Yaskawa INFORM job: SKRZYNIA_5540_90_STOPNI_10BR.JBI

/JOB
//NAME SKRZYNIA_5540_90_STOPNI_10BR
///FOLDERNAME 02-SKRZYNIE_JOBS
//POS
///NPOS 687,687,0,50,0,0
///TOOL 0
///POSTYPE PULSE
///PULSE
C00000=0,-52280,40443,0,6876,0
C00001=82314,-24956,17040,59626,-27382,6248
C00002=93910,-8625,17040,59626,-43355,6248
C00003=98846,-1061,-42166,80308,-57081,-16120
C00004=100452,6057,-48127,85711,-56704,-21322
C00005=96349,29000,-36127,85072,-63022,-26262
C00006=95580,33075,-33256,84644,-64024,-26851
C00007=94197,33846,-32020,85210,-63413,-26698
C00008=95580,33075,-33256,84644,-64024,-26851
C00009=94888,31114,-36362,85298,-63687,-27185
C00010=95580,33075,-33256,84644,-64024,-26851
C00011=95263,33142,-33256,84677,-63995,-26850
C00012=94634,33491,-32695,84935,-63717,-26781
C00013=94130,33776,-32235,85140,-63494,-26725
C00014=95104,32689,-33981,84829,-63917,-26928
C00015=94679,31503,-35865,85229,-63711,-27129
C00016=95263,33142,-33256,84677,-63995,-26850
C00017=95260,33144,-33256,84678,-63995,-26850
C00018=94650,33483,-32714,84929,-63727,-26783
C00019=94112,33789,-32223,85148,-63489,-26723
C00020=95084,32644,-34054,84845,-63909,-26937
C00021=94657,31449,-35950,85247,-63703,-27139
C00022=95260,33144,-33256,84678,-63995,-26850
C00023=95258,33145,-33257,84676,-63996,-26846
C00024=94953,33314,-32988,84801,-63862,-26812
C00025=94037,33833,-32158,85174,-63457,-26709
C00026=94978,32352,-34521,84941,-63860,-26983
C00027=94597,31295,-36193,85297,-63678,-27162
C00028=95258,33145,-33257,84676,-63996,-26846
C00029=95258,33145,-33257,84676,-63996,-26846
C00030=94635,33491,-32703,84932,-63720,-26777
C00031=94255,33706,-32357,85087,-63552,-26734
C00032=95076,32627,-34084,84849,-63906,-26937
C00033=94616,31344,-36119,85281,-63684,-27155
C00034=95258,33145,-33257,84676,-63996,-26846
C00035=95258,25631,32269,66559,-75499,-2416
C00036=95045,25799,32513,66531,-75379,-2372
C00037=94321,26382,33365,66429,-74973,-2219
C00038=95048,24784,31042,66584,-75290,-2483
C00039=94601,23046,28557,66633,-74859,-2609
C00040=95258,25631,32269,66559,-75499,-2416
C00041=98646,19496,-17631,99827,-80462,-21224
C00042=98317,21326,-15127,99395,-81089,-20992
C00043=97962,21529,-14845,99504,-80870,-20995
C00044=98567,20146,-16748,99341,-81286,-21080
C00045=98203,18829,-18537,99489,-81121,-21211
C00046=98811,21047,-15512,99242,-81394,-20987
C00047=98811,19937,1242,97498,-78933,-15296
C00048=98811,19937,1242,97498,-78933,-15296
C00049=98014,20416,1894,97635,-78400,-15298
C00050=98593,19084,88,97564,-78819,-15379
C00051=98194,17557,-1953,97683,-78607,-15521
C00052=98811,19937,1242,97498,-78933,-15296
C00053=98765,34858,63506,90961,-74847,-417
C00054=98962,39103,70654,91062,-76265,452
C00055=98093,40155,72476,90768,-75677,655
C00056=98962,39103,70654,91062,-76265,452
C00057=98539,36034,65455,91246,-76081,-158
C00058=98962,39103,70654,91062,-76265,452
C00059=98994,31803,58419,90917,-73461,-1055
C00060=94428,854,16076,89248,-50738,-4740
C00061=88080,-20128,-3199,80943,-31244,-2335
C00062=48287,-44591,-17414,16172,-14532,25809
C00063=48287,-44591,-17414,16172,-14532,25809
C00064=89603,-12372,12158,50295,-44413,5810
C00065=98990,20110,21695,70166,-74669,-10293
C00066=97443,24182,16559,71706,-75040,-13643
C00067=96724,24681,12603,72193,-76238,-15336
C00068=95373,25645,13977,72253,-75425,-15117
C00069=96724,24681,12603,72193,-76238,-15336
C00070=96395,23390,10778,72281,-75950,-15438
C00071=96724,24681,12603,72193,-76238,-15336
C00072=98418,23275,9051,78885,-77594,-17480
C00073=98418,23353,9846,78794,-77668,-17252
C00074=97172,24175,11002,78894,-76868,-17107
C00075=98418,23353,9846,78794,-77668,-17252
C00076=98085,21992,7947,78885,-77405,-17367
C00077=98418,23353,9846,78794,-77668,-17252
C00078=97055,28839,36684,71776,-79389,-10554
C00079=97055,28839,36684,71776,-79389,-10554
C00080=96073,29634,37879,71669,-78808,-10363
C00081=97055,28839,36684,71776,-79389,-10554
C00082=96556,26588,33346,71835,-78895,-10784
C00083=97055,28839,36684,71776,-79389,-10554
C00084=97055,28839,36684,71776,-79389,-10554
C00085=97055,28839,36684,71776,-79389,-10554
C00086=96070,29634,37881,71667,-78806,-10365
C00087=97055,28839,36684,71776,-79389,-10554
C00088=96542,26531,33264,71837,-78884,-10788
C00089=97055,28839,36684,71776,-79389,-10554
C00090=99222,23346,17795,82202,-78388,4176
C00091=99222,23346,17795,82202,-78388,4176
C00092=98198,24012,18735,82231,-77709,4276
C00093=99222,23346,17795,82202,-78388,4176
C00094=98846,21740,15549,82282,-78105,4028
C00095=99222,23346,17795,82202,-78388,4176
C00096=97305,19304,15511,100837,-75687,4760
C00097=97826,25373,24000,100195,-79238,5786
C00098=96887,26043,24967,100223,-78578,5793
C00099=97826,25373,24000,100195,-79238,5786
C00100=97448,23764,21701,100276,-79072,5588
C00101=97826,25373,24000,100195,-79238,5786
C00102=97826,25373,24000,100195,-79238,5786
C00103=97826,25373,24000,100195,-79238,5786
C00104=96843,26076,25015,100223,-78545,5791
C00105=97826,25373,24000,100195,-79238,5786
C00106=97441,23730,21652,100278,-79068,5583
C00107=97826,25373,24000,100195,-79238,5786
C00108=98604,24841,23235,100170,-79782,5786
C00109=98281,23602,18484,100238,-79492,4693
C00110=96938,24614,19922,100310,-78605,4704
C00111=98281,23602,18484,100238,-79492,4693
C00112=97922,22110,16391,100318,-79328,4520
C00113=98281,23602,18484,100238,-79492,4693
C00114=97826,25373,24000,100195,-79238,5786
C00115=100071,8792,-2363,102947,-71408,2025
C00116=90699,-12620,-30080,113827,-52438,-6201
C00117=97832,-16290,-36993,112551,-57584,-6005
C00118=83036,-26396,-56580,138157,-49269,-16960
C00119=83036,-26453,-52828,136768,-47205,-15962
C00120=60067,-65836,-77869,147206,-28305,-20439
C00121=63330,-26972,24478,18707,-56801,31483
C00122=86830,-18603,-3985,49492,-42347,15253
C00123=100465,-3562,-10252,69901,-61773,-201
C00124=99635,18997,3540,80919,-74698,-6325
C00125=98097,22561,8426,80415,-76730,-6116
C00126=98097,22561,8426,80415,-76730,-6116
C00127=97377,23028,9077,80478,-76265,-6042
C00128=98097,22561,8426,80415,-76730,-6116
C00129=97807,21406,6827,80497,-76510,-6215
C00130=98097,22561,8426,80415,-76730,-6116
C00131=98919,31293,46565,87609,-78984,1304
C00132=98899,30801,44624,87834,-79065,838
C00133=98247,31325,45433,87747,-78622,912
C00134=98899,30801,44624,87834,-79065,838
C00135=98602,29264,42279,87883,-78869,621
C00136=98899,30801,44624,87834,-79065,838
C00137=98482,30562,41503,101958,-78355,-2440
C00138=98031,30614,41582,101940,-78055,-2471
C00139=96674,31741,43313,101828,-77074,-2426
C00140=98031,30614,41582,101940,-78055,-2471
C00141=97723,29096,39278,102008,-77969,-2698
C00142=98031,30614,41582,101940,-78055,-2471
C00143=99865,12124,7354,104364,-73625,-7862
C00144=80898,-21381,-5865,68721,-28456,7693
C00145=53207,-50775,-37673,21053,-11333,28727
C00146=44299,-51091,-32799,-7549,-14278,41753
///LIMIT ON
C00147=42754,-66126,12236,-1301,3231,7194
///LIMIT OFF
C00148=0,-52280,40443,0,6876,0
C00149=0,-52280,40443,0,6876,0
C00150=0,-43112,23163,-32261,-40956,-29092
C00151=48283,-21883,28214,25170,-26491,-48363
C00152=46664,-3144,58041,18842,-32105,-45325
C00153=50347,-18571,12268,49104,-16423,-60029
C00154=51149,-18702,10839,52647,-16284,-61663
C00155=49023,-16654,12458,50505,-14948,-60880
C00156=50458,-16314,12735,52976,-15639,-61913
C00157=50509,-19000,10610,51503,-15997,-61182
C00158=50509,-19000,10610,51503,-15997,-61182
C00159=51153,-18191,11234,52953,-16222,-61812
C00160=49506,-16603,12499,51322,-15186,-61219
C00161=50699,-16390,12671,53298,-15774,-62041
C00162=50704,-18403,11069,52157,-16018,-61478
C00163=50704,-18403,11069,52157,-16018,-61478
C00164=51011,-18259,11181,52703,-16157,-61707
C00165=49372,-16676,12437,51065,-15128,-61110
C00166=50855,-16321,12727,53567,-15849,-62152
C00167=50704,-18403,11069,52157,-16018,-61478
C00168=50704,-18403,11069,52157,-16018,-61478
C00169=51194,-17966,11787,52443,-16367,-61556
C00170=49641,-16469,12982,50879,-15396,-60984
C00171=51159,-16110,13274,53409,-16135,-62034
C00172=51194,-19029,8982,55593,-15729,-63095
C00173=51005,-17995,11387,52847,-16122,-61778
C00174=51030,-17982,11395,52891,-16135,-61798
C00175=49666,-16664,12446,51542,-15278,-61306
C00176=51234,-16283,12753,54139,-16047,-62382
C00177=51030,-17982,11395,52891,-16135,-61798
C00178=51030,-17982,11395,52891,-16135,-61798
C00179=51056,-17951,11420,52949,-16145,-61823
C00180=49507,-16445,12622,51407,-15172,-61259
C00181=51212,-15994,12989,54262,-16005,-62444
C00182=51056,-17951,11420,52949,-16145,-61823
C00183=50945,-18019,11363,52741,-16103,-61737
C00184=51451,-18380,9957,55416,-15976,-62984
C00185=49638,-16617,11364,53777,-14815,-62399
C00186=51249,-16205,11700,56405,-15635,-63491
C00187=50945,-18019,11363,52741,-16103,-61737
C00188=50945,-18019,11363,52741,-16103,-61737
C00189=51751,-18888,8325,57986,-15754,-64205
C00190=49901,-17096,9744,56519,-14545,-63700
C00191=51443,-16713,10055,58931,-15359,-64698
C00192=50945,-18019,11363,52741,-16103,-61737
C00193=50945,-18019,11363,52741,-16103,-61737
C00194=51752,-17629,11670,54137,-16475,-62321
C00195=49778,-15710,13222,52239,-15234,-61634
C00196=51536,-15216,13634,55124,-16102,-62830
C00197=50945,-18019,11363,52741,-16103,-61737
C00198=50028,-22953,-3957,22347,-31919,-54220
C00199=50556,-22259,-3444,23037,-31901,-54554
C00200=48685,-20311,-1961,21193,-31011,-53711
C00201=50316,-19877,-1623,23110,-31344,-54618
C00202=49456,-22793,-3840,21729,-31736,-53932
C00203=49763,-25421,-36239,24565,-26935,-60445
C00204=49763,-25421,-36239,24565,-26935,-60445
C00205=47682,-22631,-34091,22709,-25786,-59390
C00206=49411,-21994,-33587,24802,-26153,-60557
C00207=49763,-25421,-36239,24565,-26935,-60445
C00208=50713,-12366,-58367,41124,-17813,-74400
C00209=50531,-11018,-57111,41258,-17631,-74434
C00210=49339,-9106,-55286,40470,-17030,-73839
C00211=50327,-8799,-54988,41498,-17395,-74518
C00212=50078,-11370,-57441,40744,-17481,-74102
C00213=49763,-25421,-36239,24565,-26935,-60445
C00214=49426,-25689,-5908,21254,-32432,-53672
C00215=45389,-28224,4312,35967,-15579,-54278
C00216=40154,-51179,-915,24203,-8234,-36524
C00217=0,-52280,40443,0,6876,0
C00218=0,-52280,40443,0,6876,0
C00219=2117,-50103,-33543,4117,45077,-85249
C00220=-26439,-48928,-33543,4117,-52362,-85249
C00221=-26439,-27355,-33543,41485,-52362,-85249
C00222=-47486,-18593,-22655,32887,-41344,-78763
C00223=-48804,2873,-12100,24189,-42468,-81113
C00224=-46457,7101,-11330,26648,-40775,-82885
C00225=-47278,8641,-9483,26175,-40625,-82510
C00226=-46717,9819,-8044,26408,-40882,-82710
C00227=-47278,8641,-9483,26175,-40625,-82510
C00228=-48464,9694,-8203,25521,-40353,-81986
C00229=-47278,8641,-9483,26175,-40625,-82510
C00230=-44522,-635,-31983,49264,-28311,-89687
C00231=-44904,-149,-31453,49090,-28120,-89538
C00232=-44398,873,-30329,49324,-28371,-89731
C00233=-44904,-149,-31453,49090,-28120,-89538
C00234=-45751,485,-30759,48680,-27706,-89207
C00235=-44904,-149,-31453,49090,-28120,-89538
C00236=-41365,-13075,-22481,51159,-38446,-84131
C00237=-20796,-2039,-9686,94158,-57077,-89438
C00238=-24380,-971,-8542,94589,-54660,-89617
C00239=-25651,-542,-8077,94748,-53804,-89683
C00240=-25378,473,-6965,94714,-53986,-89667
C00241=-25651,-542,-8077,94748,-53804,-89683
C00242=-26467,-222,-7729,94854,-53254,-89725
C00243=-25651,-542,-8077,94748,-53804,-89683
C00244=-25651,-542,-8077,94748,-53804,-89683
C00245=-25946,-428,-7954,94785,-53605,-89698
C00246=-25690,517,-6922,94753,-53778,-89686
C00247=-25946,-428,-7954,94785,-53605,-89698
C00248=-26504,-206,-7715,94856,-53230,-89728
C00249=-25946,-428,-7954,94785,-53605,-89698
C00250=-4522,-31762,-35329,90790,-67707,-86470
C00251=34878,-25684,-31064,90205,-94657,-86497
C00252=34878,-25684,-31064,90205,-94657,-86497
C00253=-29329,5838,20653,63819,-53216,-67184
C00254=-29329,5838,20653,63819,-53216,-67184
C00255=-29048,6776,21767,63865,-53412,-67197
C00256=-29329,5838,20653,63819,-53216,-67184
C00257=-29728,6023,20871,63686,-52977,-67114
C00258=-29329,5838,20653,63819,-53216,-67184
C00259=-26603,-1578,11750,66889,-51946,-68995
C00260=-28084,-8635,-16421,94802,-52116,-89609
C00261=-26816,-2974,-10680,94869,-53013,-89721
C00262=-26345,-658,-8205,94838,-53336,-89719
C00263=-26015,535,-6901,94796,-53558,-89702
C00264=-26345,-658,-8205,94838,-53336,-89719
C00265=-26668,-531,-8065,94879,-53120,-89737
C00266=-26345,-658,-8205,94838,-53336,-89719
C00267=-25886,-767,-8323,94779,-53646,-89696
C00268=-25886,-767,-8323,94779,-53646,-89696
C00269=-25568,389,-7061,94741,-53858,-89681
C00270=-25886,-767,-8323,94779,-53646,-89696
C00271=-26674,-459,-7988,94881,-53115,-89738
C00272=-25886,-767,-8323,94779,-53646,-89696
C00273=-25886,-767,-8323,94779,-53646,-89696
C00274=-26039,-1319,-8919,94795,-53542,-89701
C00275=-25594,308,-7149,94744,-53844,-89683
C00276=-26039,-1319,-8919,94795,-53542,-89701
C00277=-26964,-954,-8527,94912,-52922,-89753
C00278=-26039,-1319,-8919,94795,-53542,-89701
C00279=-6422,-16748,-12987,81781,-66398,-84181
C00280=26295,-11282,7080,74868,-91255,-82094
C00281=26295,-11282,7080,74868,-91255,-82094
C00282=-19602,460,18931,65728,-61929,-78089
C00283=-27549,8936,28821,63115,-57256,-76757
C00284=-27549,8936,28821,63115,-57256,-76757
C00285=-27137,10499,30762,63159,-57570,-76739
C00286=-27549,8936,28821,63115,-57256,-76757
C00287=-28395,9323,29301,62815,-56766,-76608
C00288=-27549,8936,28821,63115,-57256,-76757
C00289=-25830,8846,34722,70907,-56519,-75926
C00290=-26000,11892,38571,70638,-56518,-75722
C00291=-25623,13478,40636,70627,-56817,-75642
C00292=-26000,11892,38571,70638,-56518,-75722
C00293=-26799,12251,39037,70343,-56037,-75609
C00294=-26000,11892,38571,70638,-56518,-75722
C00295=-29869,-7804,-15550,96032,-46150,-90107
C00296=-30664,-6343,-14094,96248,-45630,-90223
C00297=-30266,-5205,-12941,96241,-45907,-90235
C00298=-30664,-6343,-14094,96248,-45630,-90223
C00299=-31549,-5956,-13703,96412,-45040,-90299
C00300=-30664,-6343,-14094,96248,-45630,-90223
C00301=-30881,-6301,-14053,96286,-45485,-90239
C00302=-30881,-6301,-14053,96286,-45485,-90239
C00303=-30478,-5160,-12894,96278,-45765,-90250
C00304=-30881,-6301,-14053,96286,-45485,-90239
C00305=-31620,-5975,-13722,96425,-44990,-90303
C00306=-30881,-6301,-14053,96286,-45485,-90239
C00307=-30881,-6301,-14053,96286,-45485,-90239
C00308=-30881,-6301,-14053,96286,-45485,-90239
C00309=-30447,-5069,-12799,96277,-45787,-90250
C00310=-30881,-6301,-14053,96286,-45485,-90239
C00311=-31687,-5947,-13694,96439,-44946,-90310
C00312=-30881,-6301,-14053,96286,-45485,-90239
C00313=-40108,-3695,2740,114838,-35048,-86380
C00314=-40108,-3695,2740,114838,-35048,-86380
C00315=-39569,-2580,3911,114673,-35386,-86267
C00316=-40108,-3695,2740,114838,-35048,-86380
C00317=-40792,-3300,3152,115124,-34647,-86568
C00318=-40108,-3695,2740,114838,-35048,-86380
C00319=-30881,-6301,-14053,96286,-45485,-90239
C00320=-26558,-19284,-27675,95285,-48332,-89713
C00321=-5136,-57382,-50746,80999,-31115,-81799
C00322=-5136,-57382,-50746,80999,-31115,-81799
C00323=-28081,-5880,-3448,89665,-51503,-85625
C00324=-29146,-693,14124,66641,-54461,-78263
C00325=-27186,7805,23879,67003,-55804,-78365
C00326=-27186,7805,23879,67003,-55804,-78365
C00327=-26901,8878,25190,67028,-56018,-78354
C00328=-27186,7805,23879,67003,-55804,-78365
C00329=-27820,8088,24221,66810,-55415,-78267
C00330=-27186,7805,23879,67003,-55804,-78365
C00331=-29983,12431,36540,97303,-47015,-80901
C00332=-29983,5395,14068,105725,-49606,-86937
C00333=-29614,6622,15514,105627,-49820,-86846
C00334=-29983,5395,14068,105725,-49606,-86937
C00335=-30655,5720,14449,105789,-49168,-87017
C00336=-29983,5395,14068,105725,-49606,-86937
C00337=-23275,-722,28392,94611,-50650,-77911
C00338=1657,-52280,40443,-304,6876,209
C00339=80083,-25473,16734,55938,-25627,7512
C00340=92674,-9533,16184,58080,-41894,6874
C00341=98391,-2369,-43566,80825,-55961,-16033
C00342=100022,4785,-49618,86526,-55706,-21348
C00343=95373,33537,-36121,86560,-63232,-28029
C00344=93881,36038,-32437,85059,-64562,-27761
C00345=93867,33044,-30650,83528,-64743,-25992
C00346=94930,31411,-33227,84334,-64171,-26252
C00347=94930,31411,-33227,84334,-64171,-26252
C00348=93474,31409,-33627,85103,-63552,-26381
C00349=93474,31409,-33627,85103,-63552,-26381
C00350=96539,31728,-33125,83558,-64961,-26367
C00351=95609,19235,-3385,72159,-68881,-11456
C00352=93675,20756,-1492,72153,-69304,-11461
C00353=93706,20835,-1296,72059,-69329,-11411
C00354=95041,22056,296,71883,-70234,-11460
C00355=95041,22056,296,71883,-70234,-11460
C00356=93716,20674,-1606,72153,-69328,-11471
C00357=93749,20787,-1450,72141,-69355,-11463
C00358=95041,22056,296,71883,-70234,-11460
C00359=95041,22056,296,71883,-70234,-11460
C00360=93853,20645,-1646,72134,-69414,-11487
C00361=93701,20690,-1585,72152,-69318,-11471
C00362=95606,21673,-233,71830,-70568,-11545
C00363=95936,-8790,-36169,76308,-52611,-10237
C00364=87381,-35372,-46042,66676,-50803,-1891
C00365=84950,-62287,8062,38288,-37295,1216
C00366=1657,-52280,40443,-304,6876,209
C00367=1657,-52280,40443,-304,6876,209
C00368=841,-50033,-33518,5341,45264,-86395
C00369=-28809,-48989,-33566,1638,-52261,-83793
C00370=-27557,-28108,-34083,40495,-51335,-84423
C00371=-43175,-5028,3939,29661,-52136,-76374
C00372=-47795,3485,-15813,29932,-36086,-79941
C00373=-44015,2890,-15585,39685,-35939,-88215
C00374=-42914,6338,-14016,39581,-38587,-88416
C00375=-47171,-3603,-26071,35496,-30340,-86638
C00376=-39353,-3849,1639,43041,-43888,-84310
C00377=-40294,353,6523,42392,-43585,-83914
C00378=-40294,-1845,-2536,45888,-40368,-86147
C00379=-39436,-6261,-5399,45238,-41722,-85736
C00380=-30485,-11577,-22290,99557,-44658,-90261
C00381=-27060,524,-8030,98323,-53088,-89706
C00382=-27060,2516,2295,94290,-52181,-86514
C00383=-23772,-4569,-11810,96993,-55055,-88783
C00384=4678,-17958,4683,47898,-79597,-85332
C00385=-18355,-35625,17567,22328,-38004,-35198
C00386=38277,-55351,-7622,112862,-31065,-32489
C00387=1657,-52280,40443,-304,6876,209
C00388=-4811,-36310,24637,-49210,-33845,-31988
C00389=41748,-30202,7105,17690,-22932,-42913
C00390=41748,-30202,7105,17690,-22932,-42913
C00391=49037,-21406,10886,33705,-21312,-49933
C00392=57938,-18196,5914,66765,-23183,-68504
C00393=62071,-18819,1330,80566,-26873,-76175
C00394=48249,-23742,8050,33819,-21114,-50004
C00395=-4811,-36310,24637,-49210,-33845,-31988
C00396=1657,-52280,40443,-304,6876,209
C00397=1613,-52280,40443,-296,6876,203
C00398=73560,-62084,7826,28695,-34737,3666
C00399=88377,-34186,-45291,67238,-52212,-2442
C00400=96528,-7533,-34932,76119,-53878,-10439
C00401=100432,21324,12575,83706,-77956,-7498
C00402=98573,22459,14150,83808,-76714,-7352
C00403=97684,25950,19098,83414,-79070,-7056
C00404=97598,25982,19143,83418,-79013,-7051
C00405=99338,18438,8643,84272,-74238,-7648
C00406=99336,18440,8642,84276,-74234,-7647
C00407=97786,25707,18749,83415,-79135,-7087
C00408=97740,25808,18892,83414,-79103,-7073
C00409=99336,18440,8642,84276,-74234,-7647
C00410=99336,18440,8642,84276,-74234,-7647
C00411=97857,25790,18866,83408,-79181,-7079
C00412=97666,25767,18833,83421,-79056,-7078
C00413=99336,18440,8642,84276,-74234,-7647
C00414=100441,9433,14994,80938,-68243,-1963
C00415=97304,12984,-1939,107395,-74362,-11877
C00416=95714,22990,10978,105436,-80284,-10194
C00417=95695,24324,20069,104661,-78619,-7848
C00418=97365,14710,-1887,106999,-76950,-12059
C00419=98851,2841,7216,80537,-62817,-1838
C00420=99868,-33,22146,72719,-59601,5126
C00421=99028,-10516,17309,71061,-60695,4227
C00422=58820,-39124,10926,53325,-41870,3759
C00423=0,-52280,40443,0,6876,0
C00424=37281,-50778,-9546,79570,-75313,-71156
C00425=21038,-23698,-30323,82948,-81132,-85647
C00426=7436,-16003,-3781,101119,-69483,-78457
C00427=-27121,-5377,5501,98364,-47418,-81834
C00428=-29080,8413,23722,96931,-48705,-80906
C00429=-31669,8189,15332,113614,-50161,-86745
C00430=-29309,2640,17780,96201,-45535,-80500
C00431=-23641,-6994,7554,96186,-49257,-79992
C00432=19501,-22886,-23351,116550,-78011,-79854
C00433=12194,-41912,-2470,49602,-55297,-50296
C00434=32334,-18287,-16541,87042,-89296,-82607
C00435=-25600,-16732,-29668,75447,-47301,-83964
C00436=-34326,1953,-11448,60781,-44929,-78860
C00437=-37866,4305,-6967,50208,-44378,-75448
C00438=-31045,-6665,-14727,69712,-44450,-80944
C00439=-32820,-434,4418,65374,-45715,-76243
C00440=-32820,-2501,-4362,69422,-44138,-78966
C00441=-29656,-6663,-8020,66257,-46678,-78481
C00442=-38755,-17773,-33721,67311,-34017,-81961
C00443=-35581,-11023,-27644,69090,-35721,-83210
C00444=-30590,527,-16574,72341,-46994,-87004
C00445=-30590,212,-22171,75529,-46132,-89216
C00446=-33949,-22068,-37275,67306,-37324,-82274
C00447=-40042,-68802,-18337,47708,-19461,-45384
C00448=-37287,-55159,35520,2191,5667,-2084
C00449=0,-52280,40443,0,6876,0
C00450=0,-36700,24612,-42871,-31823,-33862
C00451=44403,-30110,7154,24155,-23805,-45557
C00452=48366,-23967,9999,33441,-23050,-49710
C00453=57059,-21871,4355,62840,-24072,-66406
C00454=62606,-18539,1219,81479,-27911,-78168
C00455=65882,-18177,-2494,91427,-32157,-83791
C00456=50677,-23266,8367,38735,-22212,-52049
C00457=47073,-34549,9488,27883,-30316,-51458
C00458=0,-52280,40443,0,6876,0
C00459=0,-52280,40443,0,6876,0
C00460=73560,-62084,7826,28695,-34737,3666
C00461=87376,-41373,-10333,58133,-51016,401
C00462=100341,-12426,-15111,78591,-60044,-5220
C00463=100467,-7393,-15195,81625,-60158,-6002
C00464=99336,18440,8642,84276,-74234,-7647
C00465=98831,26826,38209,85264,-77545,-1440
C00466=97968,30695,40017,90402,-79732,-2682
C00467=98020,30578,39840,90409,-79769,-2698
C00468=101143,13060,5845,92851,-72534,-7825
C00469=100831,4438,-8389,94728,-68210,-9698
C00470=98542,-16618,-45693,112471,-63837,-17484
C00471=88321,-38303,-37571,90324,-45217,-1978
C00472=73315,-17786,32032,37482,-51892,27783
C00473=73315,-17786,32032,37482,-51892,27783
C00474=93279,7912,57349,51328,-58559,22694
C00475=99912,22097,29813,73010,-76799,4238
C00476=97600,19185,18425,74160,-73885,1810
C00477=96784,28529,39151,73372,-79002,4715
C00478=96741,24771,24035,74701,-77176,1243
C00479=98434,25220,35553,73286,-78430,4793
C00480=96935,989,20209,68430,-59885,10515
C00481=79425,-37128,-15462,51820,-35721,18807
C00482=43180,-50572,-20637,6552,-29302,38834
///LIMIT ON
C00483=37721,-67612,11381,1325,-438,7850
///LIMIT OFF
C00484=-37287,-55159,35520,2191,5667,-2084
C00485=-40042,-68802,-18337,47708,-19461,-45384
C00486=-28646,-23138,-32952,89786,-42552,-85395
C00487=-30193,-12825,-24186,91372,-43752,-86505
C00488=-31120,-5451,-17038,91814,-44683,-86873
C00489=-31134,-5488,-17074,91814,-44673,-86872
C00490=-30706,-9539,-21090,91641,-44141,-86712
C00491=-30706,-9539,-21090,91641,-44141,-86712
C00492=-33095,-7143,-18859,92591,-41579,-87147
C00493=-33112,-7185,-18903,92591,-41567,-87145
C00494=-33746,-1176,10845,101603,-40605,-81585
C00495=-10974,-25157,-10641,98520,-54806,-77487
C00496=31369,-21210,-7704,102203,-82608,-74705
C00497=31369,-21210,-7704,102203,-82608,-74705
C00498=32236,-17736,2151,73206,-90006,-78496
C00499=2413,-16607,2080,65101,-71431,-76259
C00500=-34840,2394,22974,48249,-51640,-69452
C00501=-33831,18589,49739,44880,-63097,-61844
C00502=-33831,13710,36104,47061,-59222,-64049
C00503=-35408,1628,18221,49605,-49628,-70543
C00504=-36029,-1090,16876,49320,-48191,-69422
C00505=-45963,-23918,13188,27154,-34733,-49172
C00506=0,-52280,40443,0,6876,0
C00507=37164,-60659,6466,13301,-5027,-19773
C00508=45362,-39990,2831,27538,-17767,-40935
C00509=55315,-20486,12421,43917,-25084,-54085
C00510=61760,-17076,4399,78300,-26495,-75523
C00511=66887,-15221,5723,82563,-32969,-76938
C00512=53534,-30170,6270,37667,-26637,-51098
C00513=41180,-61187,4729,17280,-8498,-23442
C00514=0,-52280,40443,0,6876,0
C00515=0,-52280,40443,0,6876,0
///LIMIT ON
C00516=37721,-67612,11381,1325,-438,7850
///LIMIT OFF
C00517=43180,-50572,-20637,6552,-29302,38834
C00518=79425,-37128,-15462,51820,-35721,18807
C00519=93780,-25751,-26111,76451,-39821,4971
C00520=100090,6189,-451,83287,-67207,-856
C00521=99662,22785,17568,82066,-77607,-1267
C00522=98003,26711,23176,81782,-79695,-932
C00523=98187,26766,23256,81772,-79821,-932
C00524=99662,22785,17568,82066,-77607,-1267
C00525=99662,22785,17568,82066,-77607,-1267
C00526=97671,26258,22515,81825,-79282,-965
C00527=97727,26283,22551,81822,-79321,-966
C00528=99662,22785,17568,82066,-77607,-1267
C00529=99662,22785,17568,82066,-77607,-1267
C00530=97804,25700,21708,81856,-79094,-1026
C00531=97599,25610,21578,81868,-78954,-1030
C00532=99662,22785,17568,82066,-77607,-1267
C00533=97206,-2526,-13508,84298,-60212,-1778
C00534=99581,-17537,-27968,84120,-53285,-833
C00535=87335,-30812,-23405,71152,-48070,8074
C00536=43180,-50572,-20637,6552,-29302,38834
///LIMIT ON
C00537=37721,-67612,11381,1325,-438,7850
///LIMIT OFF
C00538=0,-52280,40443,0,6876,0
C00539=0,-52280,40443,0,6876,0
C00540=-37287,-55159,35520,2191,5667,-2084
C00541=-40042,-68802,-18337,47708,-19461,-45384
C00542=-46318,-50945,-29177,106898,-20771,-78142
C00543=-46775,-41793,-28600,116864,-25974,-84568
C00544=-37035,-31234,-22655,117900,-33576,-84505
C00545=-33623,-10331,-13330,109256,-42555,-87094
C00546=-33459,-4510,-9104,107028,-43857,-87640
C00547=-36854,1758,5452,119173,-43239,-89918
C00548=-43373,7690,30281,135695,-33936,-89271
C00549=-40042,-68802,-18337,47708,-19461,-45384
C00550=-37287,-55159,35520,2191,5667,-2084
C00551=0,-52280,40443,0,6876,0
C00552=0,-52280,40443,0,-40770,0
C00553=-67457,-24715,25918,-9670,-26808,-27227
C00554=-30973,4607,39277,65194,-48165,-66059
C00555=-30235,-3513,14627,74857,-45278,-72652
C00556=-26454,5967,16213,83262,-53276,-77946
C00557=-26493,9871,28974,79170,-53890,-74636
C00558=-27720,3034,27192,73868,-49997,-71314
C00559=-30973,4607,39277,65194,-48165,-66059
C00560=-26978,21042,61188,69162,-56646,-66182
C00561=-27057,36371,96164,62501,-61356,-59953
C00562=-30973,4607,39277,65194,-48165,-66059
C00563=-35251,-18143,20376,53513,-41117,-59413
C00564=-9534,-43450,13514,26959,-29486,-38723
C00565=-22834,-59963,22946,6692,-2150,-9612
C00566=0,-52280,40443,0,6876,0
///LIMIT ON
C00567=23708,-46776,23536,16027,-4787,-19738
///LIMIT OFF
C00568=50917,-40459,4132,34421,-18173,-42391
C00569=55315,-20486,12421,43917,-25084,-54085
C00570=52021,-27344,-11614,25442,-32756,-51822
C00571=62388,-19076,-7315,47741,-37100,-57915
C00572=60492,-23043,-43968,60514,-28343,-68592
C00573=52021,-27344,-11614,25442,-32756,-51822
C00574=46096,-45842,-2681,20981,-19497,-36310
C00575=41180,-61187,4729,17280,-8498,-23442
C00576=0,-52280,40443,0,6876,0
C00577=0,-52280,40443,0,6876,0
///LIMIT ON
C00578=37721,-67612,11381,1325,-438,7850
///LIMIT OFF
C00579=43180,-50572,-20637,6552,-29302,38834
C00580=89824,-18072,-2764,64157,-38856,12549
C00581=98203,16433,5975,106740,-76906,-7461
C00582=95380,23681,15858,105888,-79485,-6352
C00583=95372,23687,15868,105888,-79480,-6352
C00584=95494,24167,16550,105816,-79738,-6257
C00585=95392,24052,16387,105831,-79681,-6279
C00586=95324,24045,16377,105840,-79638,-6287
C00587=98203,16433,5975,106740,-76906,-7461
C00588=100438,3826,-9542,108367,-72171,-8932
C00589=98957,-20219,-27813,100777,-56896,-5666
C00590=87335,-30812,-23405,71152,-48070,8074
C00591=80632,-38079,-20908,64053,-45216,12949
C00592=43180,-50572,-20637,6552,-29302,38834
///LIMIT ON
C00593=37721,-67612,11381,1325,-438,7850
///LIMIT OFF
C00594=0,-52280,40443,0,6876,0
C00595=-54026,-30203,28811,-7745,-28969,-5087
C00596=-81492,-18979,22896,-11682,-23662,-26316
C00597=-31639,1998,34377,78496,-41866,-64115
C00598=-28167,19375,56310,81342,-50085,-63750
C00599=-28167,28622,78575,74894,-51467,-58871
C00600=-33078,8378,41935,77523,-41039,-63739
C00601=-46905,3098,9726,144001,-39915,-89043
C00602=-37647,13740,22660,131317,-50520,-79512
C00603=-37647,16845,33202,128344,-47106,-77354
C00604=-46905,3098,9726,144001,-39915,-89043
C00605=-42864,18028,43807,131618,-37529,-87119
C00606=-44052,21146,48203,131480,-36504,-87179
C00607=-44605,22126,50160,132440,-35973,-87409
C00608=-42864,18028,43807,131618,-37529,-87119
C00609=-32723,6704,21658,111173,-45396,-82543
C00610=-34422,-9999,20796,72411,-42519,-66994
C00611=-35251,-18143,20376,53513,-41117,-59413
C00612=-9534,-43450,13514,26959,-29486,-38723
C00613=-22834,-59963,22946,6692,-2150,-9612
C00614=0,-52280,40443,0,6876,0
///LIMIT ON
C00615=23708,-46776,23536,16027,-4787,-19738
///LIMIT OFF
C00616=50917,-40459,4132,34421,-18173,-42391
C00617=56351,-28617,-8977,50177,-24220,-59041
C00618=61013,-25727,-20437,91852,-25479,-87385
C00619=68741,-23000,-19911,95900,-36007,-87783
C00620=59870,-32730,-20784,77712,-26701,-76039
C00621=36994,-41399,-15582,14937,-21377,-43241
C00622=31287,-69981,-10850,7253,-6843,-20996
C00623=19644,-57271,30737,863,5243,-2499
C00624=0,-52280,40443,0,6876,0
C00625=0,-52280,40443,0,6876,0
///LIMIT ON
C00626=37721,-67612,11381,1325,-438,7850
///LIMIT OFF
C00627=43180,-50572,-20637,6552,-29302,38834
C00628=91491,-24684,-21166,88739,-36252,3466
C00629=97242,3374,-16308,110175,-70668,-7391
C00630=94438,9043,11685,105132,-63464,-738
C00631=95457,24391,34083,103168,-72837,2707
C00632=95457,28954,48844,101249,-71049,5851
C00633=97758,10009,10083,105270,-68443,-874
C00634=95862,-16818,-21974,111833,-51241,-5826
C00635=73375,-46579,-48123,122197,-29369,-11841
C00636=61510,-42696,-20641,91785,-15812,2767
C00637=61510,-42696,-20641,91785,-15812,2767
C00638=91998,2716,51200,51967,-51421,19589
C00639=99547,21785,17244,85875,-76675,-945
C00640=97758,24649,21282,85635,-78482,-675
C00641=97758,26167,28392,84986,-78619,1092
C00642=99547,21785,17244,85875,-76675,-945
C00643=98541,21134,18604,96699,-76883,-2153
C00644=97093,25194,24413,97463,-78486,-1748
C00645=97108,27415,33780,96610,-77663,471
C00646=100501,23939,19565,97610,-81211,-2656
C00647=100157,21698,27046,96662,-76573,223
C00648=100157,21698,27046,96662,-76573,223
C00649=97571,28800,39823,95486,-77298,2019
C00650=94718,27212,28935,108231,-77656,-3237
C00651=97525,24074,14749,108994,-82208,-6125
C00652=100589,15292,8687,99532,-76329,-3922
C00653=96009,-5298,2682,83996,-53338,4019
C00654=96357,-12578,4213,73824,-49473,9415
C00655=89302,-6859,38894,49988,-60910,21081
C00656=68865,-35989,-5252,49829,-38105,21179
C00657=80632,-38079,-20908,64053,-45216,12949
C00658=43180,-50572,-20637,6552,-29302,38834
C00659=37721,-67612,11381,1325,-438,7850
C00660=0,-52280,40443,0,6876,0
C00661=0,-52278,40443,0,6872,5
C00662=0,-52278,40443,31822,-65283,-46097
C00663=-7673,2330,44178,76838,-66870,-70196
C00664=-24298,4331,21590,82032,-53834,-78397
C00665=-25355,11978,31101,81910,-55720,-77904
C00666=-25359,16324,43774,78452,-56416,-74915
C00667=-24298,4331,21590,82032,-53834,-78397
C00668=-27399,765,3050,75729,-52022,-82033
C00669=-28032,2265,2084,76986,-51244,-83010
C00670=-28018,515,-6740,80640,-50528,-85787
C00671=-24993,-2283,-4754,78157,-53063,-83953
C00672=3014,-20441,-7349,104591,-68614,-79454
C00673=17388,-18739,-2459,99831,-77693,-75560
C00674=13238,-21720,-1359,93359,-59492,-72612
C00675=-10261,-46634,14475,36899,-22136,-31570
C00676=-22834,-59963,22946,6692,-2150,-9612
C00677=0,-52280,40443,0,6876,0
C00678=23708,-46776,23536,16027,-4787,-19738
C00679=50917,-40459,4132,34421,-18173,-42391
C00680=55315,-20486,12421,43917,-25084,-54085
C00681=52609,-18323,14042,41333,-23544,-53138
C00682=70054,-15959,-1295,94448,-37577,-86566
C00683=61757,-17157,6384,73937,-27308,-72117
C00684=37618,-28118,7425,14704,-21495,-41826
C00685=31287,-69981,-10850,7253,-6843,-20996
C00686=0,-52280,40443,0,6876,0
BC00000=483637
BC00001=460491
BC00002=460491
BC00003=460491
BC00004=460491
BC00005=460491
BC00006=460491
BC00007=460491
BC00008=460491
BC00009=460491
BC00010=460491
BC00011=506593
BC00012=506593
BC00013=506593
BC00014=506593
BC00015=506593
BC00016=506593
BC00017=552803
BC00018=552803
BC00019=552803
BC00020=552803
BC00021=552803
BC00022=552803
BC00023=598907
BC00024=598907
BC00025=598907
BC00026=598907
BC00027=598907
BC00028=598907
BC00029=621955
BC00030=621955
BC00031=621955
BC00032=621955
BC00033=621955
BC00034=621955
BC00035=574754
BC00036=574754
BC00037=574754
BC00038=574754
BC00039=574754
BC00040=574754
BC00041=620864
BC00042=620864
BC00043=620864
BC00044=620864
BC00045=620864
BC00046=620864
BC00047=620864
BC00048=620864
BC00049=620864
BC00050=620864
BC00051=620864
BC00052=620864
BC00053=619616
BC00054=619616
BC00055=619616
BC00056=619616
BC00057=619616
BC00058=619616
BC00059=619616
BC00060=619616
BC00061=619616
BC00062=619616
BC00063=753230
BC00064=753195
BC00065=771362
BC00066=771362
BC00067=771362
BC00068=771362
BC00069=771362
BC00070=771362
BC00071=771362
BC00072=780850
BC00073=780850
BC00074=780850
BC00075=780850
BC00076=780850
BC00077=780850
BC00078=798636
BC00079=798636
BC00080=798636
BC00081=798636
BC00082=798636
BC00083=798636
BC00084=821724
BC00085=821724
BC00086=821724
BC00087=821724
BC00088=821724
BC00089=821724
BC00090=858551
BC00091=858551
BC00092=858551
BC00093=858551
BC00094=858551
BC00095=858551
BC00096=864565
BC00097=864565
BC00098=864565
BC00099=864565
BC00100=864565
BC00101=864565
BC00102=887605
BC00103=887605
BC00104=887605
BC00105=887605
BC00106=887605
BC00107=887605
BC00108=887605
BC00109=916466
BC00110=916466
BC00111=916466
BC00112=916466
BC00113=916466
BC00114=887605
BC00115=887605
BC00116=887605
BC00117=887605
BC00118=887605
BC00119=887605
BC00120=887605
BC00121=982705
BC00122=1000911
BC00123=976590
BC00124=976734
BC00125=976734
BC00126=976734
BC00127=976734
BC00128=976734
BC00129=976734
BC00130=976734
BC00131=995300
BC00132=988419
BC00133=988419
BC00134=988419
BC00135=988419
BC00136=988419
BC00137=1050802
BC00138=1050802
BC00139=1050742
BC00140=1050802
BC00141=1050802
BC00142=1050802
BC00143=1050802
BC00144=1010233
BC00145=1011507
BC00146=951360
BC00147=873120
BC00148=827154
BC00149=827154
BC00150=827156
BC00151=935062
BC00152=935062
BC00153=964364
BC00154=966461
BC00155=966461
BC00156=966461
BC00157=966461
BC00158=904985
BC00159=904985
BC00160=904985
BC00161=904985
BC00162=904985
BC00163=843543
BC00164=843543
BC00165=843543
BC00166=843543
BC00167=843543
BC00168=782113
BC00169=782113
BC00170=782113
BC00171=782113
BC00172=782113
BC00173=720711
BC00174=720711
BC00175=720711
BC00176=720711
BC00177=720711
BC00178=662549
BC00179=662549
BC00180=662549
BC00181=662549
BC00182=662549
BC00183=597825
BC00184=597825
BC00185=597825
BC00186=597825
BC00187=597825
BC00188=536353
BC00189=536353
BC00190=536353
BC00191=536353
BC00192=536353
BC00193=474901
BC00194=474901
BC00195=474901
BC00196=474901
BC00197=474901
BC00198=474905
BC00199=474905
BC00200=474905
BC00201=474905
BC00202=474905
BC00203=474905
BC00204=474905
BC00205=474905
BC00206=474905
BC00207=474905
BC00208=474905
BC00209=474905
BC00210=474905
BC00211=474905
BC00212=474905
BC00213=474905
BC00214=474905
BC00215=474901
BC00216=548577
BC00217=548577
BC00218=492150
BC00219=423885
BC00220=423885
BC00221=423885
BC00222=493160
BC00223=493160
BC00224=493160
BC00225=493160
BC00226=493160
BC00227=493160
BC00228=493160
BC00229=493160
BC00230=539180
BC00231=539180
BC00232=539180
BC00233=539180
BC00234=539180
BC00235=539180
BC00236=495049
BC00237=485388
BC00238=485384
BC00239=485384
BC00240=485384
BC00241=485384
BC00242=485384
BC00243=485384
BC00244=508449
BC00245=508449
BC00246=508449
BC00247=508449
BC00248=508449
BC00249=508449
BC00250=485386
BC00251=485386
BC00252=600790
BC00253=562212
BC00254=562212
BC00255=562212
BC00256=562212
BC00257=562212
BC00258=562212
BC00259=563312
BC00260=600589
BC00261=600589
BC00262=600589
BC00263=600589
BC00264=600589
BC00265=600589
BC00266=600589
BC00267=623637
BC00268=623637
BC00269=623637
BC00270=623637
BC00271=623637
BC00272=623637
BC00273=669704
BC00274=669704
BC00275=669704
BC00276=669704
BC00277=669704
BC00278=669704
BC00279=658366
BC00280=643307
BC00281=740888
BC00282=738443
BC00283=715786
BC00284=715786
BC00285=715785
BC00286=715786
BC00287=715786
BC00288=715786
BC00289=715786
BC00290=715786
BC00291=715786
BC00292=715786
BC00293=715786
BC00294=715786
BC00295=784942
BC00296=784942
BC00297=784942
BC00298=784942
BC00299=784942
BC00300=784942
BC00301=807985
BC00302=807985
BC00303=807985
BC00304=807985
BC00305=807985
BC00306=807985
BC00307=854090
BC00308=854090
BC00309=854090
BC00310=854090
BC00311=854090
BC00312=854090
BC00313=854090
BC00314=854090
BC00315=854090
BC00316=854090
BC00317=854090
BC00318=854090
BC00319=854090
BC00320=854090
BC00321=854090
BC00322=990684
BC00323=984461
BC00324=984658
BC00325=984658
BC00326=984658
BC00327=984658
BC00328=984658
BC00329=984658
BC00330=984658
BC00331=969297
BC00332=969297
BC00333=969297
BC00334=969297
BC00335=969297
BC00336=969297
BC00337=940619
BC00338=460491
BC00339=460491
BC00340=460491
BC00341=460491
BC00342=460491
BC00343=460491
BC00344=460491
BC00345=461083
BC00346=461083
BC00347=499491
BC00348=507634
BC00349=497118
BC00350=507634
BC00351=488608
BC00352=496344
BC00353=488608
BC00354=496345
BC00355=534696
BC00356=542404
BC00357=534696
BC00358=534696
BC00359=557764
BC00360=565440
BC00361=557764
BC00362=557568
BC00363=557568
BC00364=557568
BC00365=557568
BC00366=557568
BC00367=492150
BC00368=423885
BC00369=423885
BC00370=423885
BC00371=423885
BC00372=481098
BC00373=480936
BC00374=480936
BC00375=480936
BC00376=477599
BC00377=477599
BC00378=477599
BC00379=477599
BC00380=477599
BC00381=477599
BC00382=477599
BC00383=477599
BC00384=477799
BC00385=477799
BC00386=477799
BC00387=508521
BC00388=598171
BC00389=670543
BC00390=670543
BC00391=670543
BC00392=670543
BC00393=732003
BC00394=732003
BC00395=598171
BC00396=508521
BC00397=509831
BC00398=557568
BC00399=557568
BC00400=606305
BC00401=559125
BC00402=559125
BC00403=566889
BC00404=559125
BC00405=566815
BC00406=605185
BC00407=612943
BC00408=605243
BC00409=605185
BC00410=628234
BC00411=636027
BC00412=628307
BC00413=628234
BC00414=628234
BC00415=694737
BC00416=694737
BC00417=694737
BC00418=694737
BC00419=643398
BC00420=611390
BC00421=599778
BC00422=599778
BC00423=599778
BC00424=542360
BC00425=521200
BC00426=436412
BC00427=459757
BC00428=459757
BC00429=459757
BC00430=459757
BC00431=427483
BC00432=427483
BC00433=589614
BC00434=592276
BC00435=597260
BC00436=597260
BC00437=597260
BC00438=598004
BC00439=598004
BC00440=598004
BC00441=598004
BC00442=650931
BC00443=650931
BC00444=658595
BC00445=658595
BC00446=658595
BC00447=620193
BC00448=620193
BC00449=620193
BC00450=828164
BC00451=903144
BC00452=909055
BC00453=912895
BC00454=916323
BC00455=977748
BC00456=977748
BC00457=868420
BC00458=557568
BC00459=557568
BC00460=557568
BC00461=547647
BC00462=598645
BC00463=606305
BC00464=628234
BC00465=640756
BC00466=640756
BC00467=648520
BC00468=648520
BC00469=648520
BC00470=648520
BC00471=648520
BC00472=648520
BC00473=727380
BC00474=726208
BC00475=771684
BC00476=771684
BC00477=763810
BC00478=763810
BC00479=763810
BC00480=757308
BC00481=748464
BC00482=748464
BC00483=748464
BC00484=620193
BC00485=620193
BC00486=635598
BC00487=635598
BC00488=635598
BC00489=643271
BC00490=641590
BC00491=681683
BC00492=681683
BC00493=689331
BC00494=620239
BC00495=620239
BC00496=620239
BC00497=749060
BC00498=763078
BC00499=749658
BC00500=735414
BC00501=735414
BC00502=735414
BC00503=727742
BC00504=736137
BC00505=709811
BC00506=620193
BC00507=576903
BC00508=514129
BC00509=423257
BC00510=423252
BC00511=484758
BC00512=484758
BC00513=539526
BC00514=539526
BC00515=748464
BC00516=748464
BC00517=748464
BC00518=767992
BC00519=778901
BC00520=784600
BC00521=786785
BC00522=786785
BC00523=794540
BC00524=786785
BC00525=809865
BC00526=809865
BC00527=817545
BC00528=809865
BC00529=855959
BC00530=855959
BC00531=863679
BC00532=855959
BC00533=855959
BC00534=855959
BC00535=855959
BC00536=810658
BC00537=748464
BC00538=748464
BC00539=599778
BC00540=620193
BC00541=620193
BC00542=612942
BC00543=610379
BC00544=610379
BC00545=658993
BC00546=670151
BC00547=646716
BC00548=593346
BC00549=585637
BC00550=620193
BC00551=620193
BC00552=722068
BC00553=722068
BC00554=744765
BC00555=742336
BC00556=742336
BC00557=742336
BC00558=742336
BC00559=765388
BC00560=765388
BC00561=765388
BC00562=765388
BC00563=750104
BC00564=672725
BC00565=672725
BC00566=672725
BC00567=591438
BC00568=480519
BC00569=423257
BC00570=423257
BC00571=423257
BC00572=423257
BC00573=423257
BC00574=486807
BC00575=539526
BC00576=539526
BC00577=748464
BC00578=748464
BC00579=748464
BC00580=816577
BC00581=861381
BC00582=861381
BC00583=869157
BC00584=884405
BC00585=884405
BC00586=892197
BC00587=884405
BC00588=884405
BC00589=875508
BC00590=855959
BC00591=855959
BC00592=810658
BC00593=748464
BC00594=748464
BC00595=762701
BC00596=791880
BC00597=794999
BC00598=794999
BC00599=794999
BC00600=794999
BC00601=823302
BC00602=823302
BC00603=823302
BC00604=823302
BC00605=823302
BC00606=823302
BC00607=829334
BC00608=823302
BC00609=823302
BC00610=774095
BC00611=750104
BC00612=672725
BC00613=672725
BC00614=672725
BC00615=591438
BC00616=529042
BC00617=573331
BC00618=572765
BC00619=633915
BC00620=633853
BC00621=633763
BC00622=633763
BC00623=633763
BC00624=633763
BC00625=748464
BC00626=748464
BC00627=913145
BC00628=914163
BC00629=925561
BC00630=909418
BC00631=909418
BC00632=909418
BC00633=909418
BC00634=909418
BC00635=909418
BC00636=909418
BC00637=957640
BC00638=957640
BC00639=1008455
BC00640=1008455
BC00641=1010172
BC00642=1008455
BC00643=1008964
BC00644=1008964
BC00645=1008964
BC00646=1008964
BC00647=1008964
BC00648=1058688
BC00649=1058688
BC00650=1058688
BC00651=1058688
BC00652=1039072
BC00653=1015758
BC00654=1008455
BC00655=969498
BC00656=967683
BC00657=855959
BC00658=810658
BC00659=733103
BC00660=733103
BC00661=834980
BC00662=921533
BC00663=949466
BC00664=969584
BC00665=969584
BC00666=969584
BC00667=969584
BC00668=969584
BC00669=969584
BC00670=969584
BC00671=969584
BC00672=963295
BC00673=944127
BC00674=908449
BC00675=754884
BC00676=672725
BC00677=672725
BC00678=749842
BC00679=772042
BC00680=792000
BC00681=792000
BC00682=792000
BC00683=853356
BC00684=853356
BC00685=757643
BC00686=757643
///POSTYPE BASE
///RECTAN
///RCONF 0,0,0,0,0,0,0,0,0,0,0,0,0,0,0,0,0,0,0,0,0,0,0,0
P00006=-2.449,0.031,8.825,0.0000,0.0000,0.0000
P00058=0.000,0.000,3.000,0.0000,0.0000,0.0000
///RCONF 1,0,0,0,0,0,0,0,0,0,0,0,0,0,0,0,0,0,0,0,0,0,0,0
P00300=-0.036,-1.505,2.318,0.0000,0.0000,0.0000
///RCONF 0,0,0,0,0,0,0,0,0,0,0,0,0,0,0,0,0,0,0,0,0,0,0,0
P00301=0.005,-4.708,-4.628,0.0000,0.0000,0.0000
P00302=0.052,-2.937,-4.426,0.0000,0.0000,0.0000
P00303=-0.004,-1.437,-4.584,0.0000,0.0000,0.0000
P00304=0.028,-1.666,-4.234,0.0000,0.0000,0.0000
P00305=-0.003,-1.920,-3.501,0.0000,0.0000,0.0000
P00306=0.015,-2.252,-3.054,0.0000,0.0000,0.0000
P00307=0.019,-2.151,-5.077,0.0000,0.0000,0.0000
P00308=-0.003,-2.092,-4.888,0.0000,0.0000,0.0000
P00309=-0.040,-2.205,-4.992,0.0000,0.0000,0.0000
P00310=-0.006,-2.490,-5.925,0.0000,0.0000,0.0000
P00311=-0.007,-2.079,-5.307,0.0000,0.0000,0.0000
P00312=-0.032,2.202,-7.632,0.0000,0.0000,0.0000
///RCONF 1,0,0,0,0,0,0,0,0,0,0,0,0,0,0,0,0,0,0,0,0,0,0,0
P00313=-0.088,1.055,2.110,0.0000,0.0000,0.0000
P00314=-0.055,1.752,1.634,0.0000,0.0000,0.0000
P00315=-0.074,0.897,1.645,0.0000,0.0000,0.0000
P00316=0.009,2.112,2.075,0.0000,0.0000,0.0000
P00317=-0.015,2.781,3.126,0.0000,0.0000,0.0000
P00320=0.036,-8.131,3.008,0.0000,0.0000,0.0000
///RCONF 0,0,0,0,0,0,0,0,0,0,0,0,0,0,0,0,0,0,0,0,0,0,0,0
P00350=11.519,-0.008,1.149,0.0000,0.0000,0.0000
P00351=13.563,-0.027,-0.653,0.0000,0.0000,0.0000
P00352=13.252,-0.027,-0.827,0.0000,0.0000,0.0000
P00353=10.971,-0.082,0.776,0.0000,0.0000,0.0000
P00354=-0.024,2.508,-1.824,0.0000,0.0000,0.0000
P00355=-0.001,2.528,-1.131,0.0000,0.0000,0.0000
P00356=-0.034,2.921,-0.262,0.0000,0.0000,0.0000
P00357=0.003,3.386,-0.091,0.0000,0.0000,0.0000
P00358=0.014,3.037,-0.020,0.0000,0.0000,0.0000
P00359=-0.005,2.731,0.912,0.0000,0.0000,0.0000
P00360=-0.011,3.412,0.438,0.0000,0.0000,0.0000
P00361=0.018,3.050,1.253,0.0000,0.0000,0.0000
P00401=3.430,-0.021,1.131,0.0000,0.0000,0.0000
P00402=-0.253,1.107,3.062,0.0000,0.0000,0.0000
P00403=-3.666,-0.015,5.328,0.0000,0.0000,0.0000
///RCONF 1,0,0,0,0,0,0,0,0,0,0,0,0,0,0,0,0,0,0,0,0,0,0,0
P00404=0.029,4.189,-1.030,0.0000,0.0000,0.0000
///RCONF 0,0,0,0,0,0,0,0,0,0,0,0,0,0,0,0,0,0,0,0,0,0,0,0
P00405=2.420,0.007,1.427,0.0000,0.0000,0.0000
P00406=3.513,-0.022,0.429,0.0000,0.0000,0.0000
///RCONF 1,0,0,0,1,0,0,0,0,0,0,0,0,0,0,0,0,0,0,0,0,0,0,0
P00407=-0.029,2.348,-1.469,0.0000,0.0000,0.0000
P00408=0.010,1.346,-1.479,0.0000,0.0000,0.0000
///RCONF 1,0,0,0,0,0,0,0,0,0,0,0,0,0,0,0,0,0,0,0,0,0,0,0
P00409=-0.026,2.090,-1.483,0.0000,0.0000,0.0000
P00410=0.001,4.491,-0.583,0.0000,0.0000,0.0000
///RCONF 1,0,0,0,1,0,0,0,0,0,0,0,0,0,0,0,0,0,0,0,0,0,0,0
P00411=-0.015,3.627,0.872,0.0000,0.0000,0.0000
P00412=0.002,3.829,0.787,0.0000,0.0000,0.0000
P00413=0.046,0.107,-0.040,0.0000,0.0000,0.0000
///RCONF 1,0,0,0,0,0,0,0,0,0,0,0,0,0,0,0,0,0,0,0,0,0,0,0
P00414=0.046,0.800,0.739,0.0000,0.0000,0.0000
///RCONF 0,0,0,0,0,0,0,0,0,0,0,0,0,0,0,0,0,0,0,0,0,0,0,0
P00415=-1.781,-1.303,3.250,0.0000,0.0000,0.0000
P00416=0.027,1.119,3.078,0.0000,0.0000,0.0000
///RCONF 1,0,0,0,1,0,0,0,0,0,0,0,0,0,0,0,0,0,0,0,0,0,0,0
P00417=0.059,4.721,3.973,0.0000,0.0000,0.0000
//INST
///DATE 2025/02/19 12:32
///ATTR SC,RW
///GROUP1 RB1,BS1
NOP
CALL JOB:MOVE_INTO_TUNNEL
MOVJ C00000 BC00000 VJ=50.00
MOVJ C00001 BC00001 VJ=30.00
MOVJ C00002 BC00002 VJ=30.00
MOVL C00003 BC00003 V=333.3
MOVJ C00004 BC00004 VJ=30.00
MOVL C00005 BC00005 V=500.0
'------------------------
'W31.2
'------------------------
MOVL C00006 BC00006 V=166.7 PL=0
REFP 3 C00007 BC00007
CALL JOB:SEARCH-R1
SET P0300 P0006
SFTON P0300
MOVL C00008 BC00008 V=66.7 PL=0
REFP 3 C00009 BC00009
CALL JOB:SEARCH-R1
SET P0300 P0006
SFTON P0300
MOVL C00010 BC00010 V=166.7 PL=0
SFTOF
'------------------------
'W31.4
'------------------------
MOVL C00011 BC00011 V=666.7
MOVL C00012 BC00012 V=83.3 PL=0
REFP 3 C00013 BC00013
CALL JOB:SEARCH-R1
SET P0301 P0006
SFTON P0301
MOVL C00014 BC00014 V=166.7 PL=0
REFP 3 C00015 BC00015
CALL JOB:SEARCH-R1
SET P0301 P0006
SFTON P0301
MOVL C00016 BC00016 V=166.7 PL=0
SFTOF
'------------------------
'W31.6
'------------------------
MOVL C00017 BC00017 V=666.7
MOVL C00018 BC00018 V=83.3 PL=0
REFP 3 C00019 BC00019
CALL JOB:SEARCH-R1
SET P0302 P0006
SFTON P0302
MOVL C00020 BC00020 V=166.7 PL=0
REFP 3 C00021 BC00021
CALL JOB:SEARCH-R1
SET P0302 P0006
SFTON P0302
MOVL C00022 BC00022 V=250.0 PL=0
SFTOF
'------------------------
'W31.8
'------------------------
MOVL C00023 BC00023 V=666.7
MOVL C00024 BC00024 V=83.3 PL=0
REFP 3 C00025 BC00025
CALL JOB:SEARCH-R1
SET P0303 P0006
SFTON P0303
MOVL C00026 BC00026 V=166.7 PL=0
REFP 3 C00027 BC00027
CALL JOB:SEARCH-R1
SET P0303 P0006
SFTON P0303
MOVL C00028 BC00028 V=250.0 PL=0
SFTOF
'------------------------
'W31.9
'------------------------
MOVL C00029 BC00029 V=666.7
MOVL C00030 BC00030 V=83.3 PL=0
REFP 3 C00031 BC00031
CALL JOB:SEARCH-R1
SET P0304 P0006
SFTON P0304
MOVL C00032 BC00032 V=166.7 PL=0
REFP 3 C00033 BC00033
CALL JOB:SEARCH-R1
SET P0304 P0006
SFTON P0304
MOVL C00034 BC00034 V=250.0 PL=0
SFTOF
'------------------------
'W31.11
'------------------------
MOVL C00035 BC00035 V=666.7
MOVL C00036 BC00036 V=83.3 PL=0
REFP 3 C00037 BC00037
CALL JOB:SEARCH-R1
SET P0305 P0006
SFTON P0305
MOVL C00038 BC00038 V=166.7 PL=0
REFP 3 C00039 BC00039
CALL JOB:SEARCH-R1
SET P0305 P0006
SFTON P0305
MOVL C00040 BC00040 V=250.0 PL=0
SFTOF
'------------------------
'W31.13
'------------------------
MOVL C00041 BC00041 V=666.7
MOVL C00042 BC00042 V=166.7 PL=0
REFP 3 C00043 BC00043
CALL JOB:SEARCH-R1
SET P0306 P0006
SFTON P0306
MOVL C00044 BC00044 V=166.7 PL=0
REFP 3 C00045 BC00045
CALL JOB:SEARCH-R1
SET P0306 P0006
SFTON P0306
MOVL C00046 BC00046 V=250.0 PL=0
SFTOF
'------------------------
'W31.14
'------------------------
MOVL C00047 BC00047 V=666.7
MOVL C00048 BC00048 V=100.0 PL=0
REFP 3 C00049 BC00049
CALL JOB:SEARCH-R1
SET P0307 P0006
SFTON P0307
MOVL C00050 BC00050 V=166.7 PL=0
REFP 3 C00051 BC00051
CALL JOB:SEARCH-R1
SET P0307 P0006
SFTON P0307
MOVL C00052 BC00052 V=250.0 PL=0
SFTOF
'------------------------
'W31.16
'------------------------
MOVL C00053 BC00053 V=666.7
MOVL C00054 BC00054 V=100.0 PL=0
REFP 3 C00055 BC00055
CALL JOB:SEARCH-R1
SET P0308 P0006
SFTON P0308
MOVL C00056 BC00056 V=166.7 PL=0
REFP 3 C00057 BC00057
CALL JOB:SEARCH-R1
SET P0308 P0006
SFTON P0308
MOVL C00058 BC00058 V=250.0 PL=0
SFTOF
MOVL C00059 BC00059 V=166.7
MOVL C00060 BC00060 V=333.3
MOVL C00061 BC00061 V=666.7
MOVL C00062 BC00062 V=500.0
MOVJ C00063 BC00063 VJ=60.00
MOVL C00064 BC00064 V=833.3 PL=0
MOVL C00065 BC00065 V=500.0 PL=0
'------------------------
'W31.18
'------------------------
MOVL C00066 BC00066 V=333.3 PL=0
SFTOF
MOVL C00067 BC00067 V=166.7 PL=0
REFP 3 C00068 BC00068
CALL JOB:SEARCH-R1
SET P0309 P0006
SFTON P0309
MOVL C00069 BC00069 V=166.7 PL=0
REFP 3 C00070 BC00070
CALL JOB:SEARCH-R1
SET P0309 P0006
SFTON P0309
MOVL C00071 BC00071 V=250.0 PL=0
SFTOF
'------------------------
'W31.19
'------------------------
MOVL C00072 BC00072 V=666.7
MOVL C00073 BC00073 V=100.0 PL=0
REFP 3 C00074 BC00074
CALL JOB:SEARCH-R1
SET P0310 P0006
SFTON P0310
MOVL C00075 BC00075 V=166.7 PL=0
REFP 3 C00076 BC00076
CALL JOB:SEARCH-R1
SET P0310 P0006
SFTON P0310
MOVL C00077 BC00077 V=250.0 PL=0
SFTOF
'------------------------
'W31.21
'------------------------
MOVL C00078 BC00078 V=666.7
MOVL C00079 BC00079 V=100.0 PL=0
REFP 3 C00080 BC00080
CALL JOB:SEARCH-R1
SET P0311 P0006
SFTON P0311
MOVL C00081 BC00081 V=166.7 PL=0
REFP 3 C00082 BC00082
CALL JOB:SEARCH-R1
SET P0311 P0006
SFTON P0311
MOVL C00083 BC00083 V=250.0 PL=0
SFTOF
'------------------------
'W31.22
'------------------------
MOVL C00084 BC00084 V=666.7
MOVL C00085 BC00085 V=100.0 PL=0
REFP 3 C00086 BC00086
CALL JOB:SEARCH-R1
SET P0312 P0006
SFTON P0312
MOVL C00087 BC00087 V=166.7 PL=0
REFP 3 C00088 BC00088
CALL JOB:SEARCH-R1
SET P0312 P0006
SFTON P0312
MOVL C00089 BC00089 V=250.0 PL=0
SFTOF
'------------------------
'W31.24
'------------------------
MOVL C00090 BC00090 V=666.7
MOVL C00091 BC00091 V=100.0 PL=0
REFP 3 C00092 BC00092
CALL JOB:SEARCH-R1
SET P0313 P0006
SFTON P0313
MOVL C00093 BC00093 V=166.7 PL=0
REFP 3 C00094 BC00094
CALL JOB:SEARCH-R1
SET P0313 P0006
SFTON P0313
MOVL C00095 BC00095 V=166.7 PL=0
SFTOF
'------------------------
'W31.26
'------------------------
MOVL C00096 BC00096 V=666.7
MOVL C00097 BC00097 V=100.0 PL=0
REFP 3 C00098 BC00098
CALL JOB:SEARCH-R1
SET P0314 P0006
SFTON P0314
MOVL C00099 BC00099 V=166.7 PL=0
REFP 3 C00100 BC00100
CALL JOB:SEARCH-R1
SET P0314 P0006
SFTON P0314
MOVL C00101 BC00101 V=250.0 PL=0
SFTOF
'------------------------
'W31.27
'------------------------
MOVL C00102 BC00102 V=666.7
MOVL C00103 BC00103 V=100.0 PL=0
REFP 3 C00104 BC00104
CALL JOB:SEARCH-R1
SET P0315 P0006
SFTON P0315
MOVL C00105 BC00105 V=166.7 PL=0
REFP 3 C00106 BC00106
CALL JOB:SEARCH-R1
SET P0315 P0006
SFTON P0315
MOVL C00107 BC00107 V=250.0 PL=0
SFTOF
MOVL C00108 BC00108 V=333.3
MOVL C00109 BC00109 V=166.7
REFP 3 C00110 BC00110
CALL JOB:SEARCH-R1
SET P0316 P0006
SFTON P0316
MOVL C00111 BC00111 V=166.7 PL=0
REFP 3 C00112 BC00112
CALL JOB:SEARCH-R1
SET P0316 P0006
SFTON P0316
MOVL C00113 BC00113 V=166.7
SFTOF
MOVL C00114 BC00114 V=250.0 PL=0
MOVL C00115 BC00115 V=666.7
MOVL C00116 BC00116 V=666.7
MOVL C00117 BC00117 V=666.7
MOVL C00118 BC00118 V=666.7
MOVL C00119 BC00119 V=666.7
MOVL C00120 BC00120 V=666.7
MOVL C00121 BC00121 V=666.7
MOVL C00122 BC00122 V=583.3
COMM MOVL C00123 BC00123 V=500.0
COMM MOVL C00124 BC00124 V=333.3 PL=0
COMM '------------------------
COMM 'W31.29
COMM '------------------------
COMM MOVL C00125 BC00125 V=166.7
COMM MOVL C00126 BC00126 V=100.0 PL=0
COMM REFP 3 C00127 BC00127
COMM CALL JOB:SEARCH-R1
COMM SET P0316 P0006
COMM SFTON P0316
COMM MOVL C00128 BC00128 V=166.7 PL=0
COMM REFP 3 C00129 BC00129
COMM CALL JOB:SEARCH-R1
COMM SET P0316 P0006
COMM SFTON P0316
COMM MOVL C00130 BC00130 V=250.0 PL=0
COMM SFTOF
'------------------------
'W31.31
'------------------------
MOVL C00131 BC00131 V=666.7
MOVL C00132 BC00132 V=166.7 PL=0
REFP 3 C00133 BC00133
CALL JOB:SEARCH-R1
SET P0317 P0006
SFTON P0317
MOVL C00134 BC00134 V=166.7 PL=0
REFP 3 C00135 BC00135
CALL JOB:SEARCH-R1
SET P0317 P0006
SFTON P0317
MOVL C00136 BC00136 V=250.0 PL=0
SFTOF
'------------------------
MOVL C00137 BC00137 V=333.3
MOVL C00138 BC00138 V=166.7
REFP 3 C00139 BC00139
CALL JOB:SEARCH-R1
SET P0320 P0006
SFTON P0320
MOVL C00140 BC00140 V=166.7 PL=0
REFP 3 C00141 BC00141
CALL JOB:SEARCH-R1
SET P0320 P0006
SFTON P0320
SFTOF
MOVL C00142 BC00142 V=250.0 PL=0
'W31.32
'------------------------
MOVL C00143 BC00143 V=500.0
MOVL C00144 BC00144 V=500.0
MOVL C00145 BC00145 V=500.0
MOVL C00146 BC00146 V=666.7
MOVJ C00147 BC00147 VJ=80.00
MOVJ C00148 BC00148 VJ=80.00
MOVJ C00149 BC00149 VJ=10.00
MOVJ C00150 BC00150 VJ=50.00
MOVJ C00151 BC00151 VJ=50.00
MOVJ C00152 BC00152 VJ=40.00
MOVL C00153 BC00153 V=500.0
SFTOF
'------------------------
'W214A P
'------------------------
MOVL C00154 BC00154 V=100.0 PL=0
REFP 3 C00155 BC00155
CALL JOB:SEARCH-R1
IMOV P0058 V=11.7
SET P0350 P0006
SFTON P0350
REFP 3 C00156 BC00156
CALL JOB:SEARCH-R1
SET P0350 P0006
SFTON P0350
MOVL C00157 BC00157 V=250.0 PL=0
SFTOF
'------------------------
'W214A L
'------------------------
MOVJ C00158 BC00158 VJ=30.00
MOVL C00159 BC00159 V=100.0 PL=0
REFP 3 C00160 BC00160
CALL JOB:SEARCH-R1
IMOV P0058 V=11.7
SET P0351 P0006
SFTON P0351
REFP 3 C00161 BC00161
CALL JOB:SEARCH-R1
SET P0351 P0006
SFTON P0351
MOVL C00162 BC00162 V=250.0 PL=0
SFTOF
'------------------------
'W219A P
'------------------------
MOVJ C00163 BC00163 VJ=40.00
MOVL C00164 BC00164 V=100.0 PL=0
REFP 3 C00165 BC00165
CALL JOB:SEARCH-R1
IMOV P0058 V=11.7
SET P0352 P0006
SFTON P0352
REFP 3 C00166 BC00166
CALL JOB:SEARCH-R1
SET P0352 P0006
SFTON P0352
MOVL C00167 BC00167 V=250.0 PL=0
SFTOF
'------------------------
'W219A L
'------------------------
MOVJ C00168 BC00168 VJ=50.00
MOVL C00169 BC00169 V=166.7 PL=0
REFP 3 C00170 BC00170
CALL JOB:SEARCH-R1
IMOV P0058 V=11.7
SET P0353 P0006
SFTON P0353
REFP 3 C00171 BC00171
CALL JOB:SEARCH-R1
SET P0353 P0006
SFTON P0353
MOVL C00172 BC00172 V=250.0 PL=0
SFTOF
'------------------------
'W213A P
'------------------------
MOVJ C00173 BC00173 VJ=60.00
MOVL C00174 BC00174 V=166.7 PL=0
REFP 3 C00175 BC00175
CALL JOB:SEARCH-R1
IMOV P0058 V=11.7
SET P0354 P0006
SFTON P0354
REFP 3 C00176 BC00176
CALL JOB:SEARCH-R1
SET P0354 P0006
SFTON P0354
MOVL C00177 BC00177 V=250.0 PL=0
SFTOF
'------------------------
'W213A L
'------------------------
MOVJ C00178 BC00178 VJ=50.00
MOVL C00179 BC00179 V=166.7 PL=0
REFP 3 C00180 BC00180
CALL JOB:SEARCH-R1
IMOV P0058 V=11.7
SET P0355 P0006
SFTON P0355
REFP 3 C00181 BC00181
CALL JOB:SEARCH-R1
SET P0355 P0006
SFTON P0355
MOVL C00182 BC00182 V=250.0 PL=0
SFTOF
'------------------------
'W218A P
'------------------------
MOVJ C00183 BC00183 VJ=60.00
MOVL C00184 BC00184 V=166.7 PL=0
REFP 3 C00185 BC00185
CALL JOB:SEARCH-R1
IMOV P0058 V=11.7
SET P0356 P0006
SFTON P0356
REFP 3 C00186 BC00186
CALL JOB:SEARCH-R1
SET P0356 P0006
SFTON P0356
MOVL C00187 BC00187 V=250.0 PL=0
SFTOF
'------------------------
'W218A L
'------------------------
MOVJ C00188 BC00188 VJ=60.00
MOVL C00189 BC00189 V=166.7 PL=0
REFP 3 C00190 BC00190
CALL JOB:SEARCH-R1
IMOV P0058 V=11.7
SET P0357 P0006
SFTON P0357
REFP 3 C00191 BC00191
CALL JOB:SEARCH-R1
SET P0357 P0006
SFTON P0357
MOVL C00192 BC00192 V=250.0 PL=0
SFTOF
'------------------------
'W215A P
'------------------------
MOVJ C00193 BC00193 VJ=60.00
MOVL C00194 BC00194 V=166.7 PL=0
REFP 3 C00195 BC00195
CALL JOB:SEARCH-R1
IMOV P0058 V=11.7
SET P0358 P0006
SFTON P0358
REFP 3 C00196 BC00196
CALL JOB:SEARCH-R1
SET P0358 P0006
SFTON P0358
MOVL C00197 BC00197 V=250.0 PL=0
SFTOF
'------------------------
'W215A L
'------------------------
MOVL C00198 BC00198 V=666.7
MOVL C00199 BC00199 V=166.7 PL=0
REFP 3 C00200 BC00200
CALL JOB:SEARCH-R1
IMOV P0058 V=11.7
SET P0359 P0006
SFTON P0359
REFP 3 C00201 BC00201
CALL JOB:SEARCH-R1
SET P0359 P0006
SFTON P0359
MOVL C00202 BC00202 V=66.7 PL=0
SFTOF
'------------------------
'W217A P
'------------------------
MOVL C00203 BC00203 V=666.7
MOVL C00204 BC00204 V=166.7 PL=0
REFP 3 C00205 BC00205
CALL JOB:SEARCH-R1
IMOV P0058 V=11.7
SET P0360 P0006
SFTON P0360
REFP 3 C00206 BC00206
CALL JOB:SEARCH-R1
SET P0360 P0006
SFTON P0360
MOVL C00207 BC00207 V=250.0 PL=0
SFTOF
'------------------------
'W217A L
'------------------------
MOVL C00208 BC00208 V=666.7
MOVL C00209 BC00209 V=166.7 PL=0
REFP 3 C00210 BC00210
CALL JOB:SEARCH-R1
IMOV P0058 V=11.7
SET P0361 P0006
SFTON P0361
REFP 3 C00211 BC00211
CALL JOB:SEARCH-R1
SET P0361 P0006
SFTON P0361
MOVL C00212 BC00212 V=250.0 PL=0
SFTOF
MOVL C00213 BC00213 V=666.7
MOVL C00214 BC00214 V=833.3
MOVL C00215 BC00215 V=833.3
MOVJ C00216 BC00216 VJ=70.00
MOVJ C00217 BC00217 VJ=80.00
COMM MOVJ C00218 BC00218 VJ=50.00
COMM MOVJ C00219 BC00219 VJ=50.00
COMM MOVJ C00220 BC00220 VJ=30.00
COMM MOVJ C00221 BC00221 VJ=30.00
COMM 'KKK
COMM MOVL C00222 BC00222 V=666.7
COMM MOVL C00223 BC00223 V=666.7
COMM MOVL C00224 BC00224 V=500.0
COMM '------------------------
COMM 'W27.4
COMM '------------------------
COMM MOVL C00225 BC00225 V=100.0 PL=0
COMM REFP 3 C00226 BC00226
COMM CALL JOB:SEARCH-R1
COMM SET P0401 P0006
COMM SFTON P0401
COMM MOVL C00227 BC00227 V=166.7 PL=0
COMM REFP 3 C00228 BC00228
COMM CALL JOB:SEARCH-R1
COMM SET P0401 P0006
COMM SFTON P0401
COMM MOVL C00229 BC00229 V=250.0 PL=0
COMM SFTOF
COMM '------------------------
COMM 'W27.6
COMM '------------------------
COMM MOVL C00230 BC00230 V=666.7
COMM MOVL C00231 BC00231 V=100.0 PL=0
COMM REFP 3 C00232 BC00232
COMM CALL JOB:SEARCH-R1
COMM SET P0402 P0006
COMM SFTON P0402
COMM MOVL C00233 BC00233 V=100.0 PL=0
COMM REFP 3 C00234 BC00234
COMM CALL JOB:SEARCH-R1
COMM SET P0402 P0006
COMM SFTON P0402
COMM MOVL C00235 BC00235 V=250.0 PL=0
COMM SFTOF
COMM MOVL C00236 BC00236 V=666.7
COMM MOVL C00237 BC00237 V=666.7
COMM '------------------------
COMM 'W27.8
COMM '------------------------
COMM MOVL C00238 BC00238 V=666.7
COMM MOVL C00239 BC00239 V=166.7 PL=0
COMM REFP 3 C00240 BC00240
COMM CALL JOB:SEARCH-R1
COMM SET P0403 P0006
COMM SFTON P0403
COMM MOVL C00241 BC00241 V=166.7 PL=0
COMM REFP 3 C00242 BC00242
COMM CALL JOB:SEARCH-R1
COMM SET P0403 P0006
COMM SFTON P0403
COMM MOVL C00243 BC00243 V=250.0 PL=0
COMM SFTOF
COMM 'ZMIENNA
COMM GETE D040 P0403 (1)
COMM GETE D041 P0403 (2)
COMM GETE D042 P0403 (3)
COMM SETE P0404 (1) D040
COMM SETE P0404 (2) D041
COMM SETE P0404 (3) D042
COMM '------------------------
COMM 'W27.9
COMM '------------------------
COMM MOVL C00244 BC00244 V=333.3
COMM MOVL C00245 BC00245 V=66.7 PL=0
COMM REFP 3 C00246 BC00246
COMM CALL JOB:SEARCH-R1
COMM SET P0404 P0006
COMM SFTON P0404
COMM MOVL C00247 BC00247 V=66.7 PL=0
COMM REFP 3 C00248 BC00248
COMM CALL JOB:SEARCH-R1
COMM SET P0404 P0006
COMM SFTON P0404
COMM MOVL C00249 BC00249 V=66.7 PL=0
COMM SFTOF
COMM MOVL C00250 BC00250 V=666.7
COMM MOVL C00251 BC00251 V=666.7
COMM MOVJ C00252 BC00252 VJ=30.00
COMM '------------------------
COMM 'W27.11
COMM '------------------------
COMM MOVL C00253 BC00253 V=500.0
COMM MOVL C00254 BC00254 V=100.0 PL=0
COMM REFP 3 C00255 BC00255
COMM CALL JOB:SEARCH-R1
COMM SET P0405 P0006
COMM SFTON P0405
COMM MOVL C00256 BC00256 V=166.7 PL=0
COMM REFP 3 C00257 BC00257
COMM CALL JOB:SEARCH-R1
COMM SET P0405 P0006
COMM SFTON P0405
COMM MOVL C00258 BC00258 V=250.0 PL=0
COMM SFTOF
COMM MOVL C00259 BC00259 V=666.7
COMM '------------------------
COMM 'W27.13
COMM '------------------------
COMM MOVL C00260 BC00260 V=666.7
COMM MOVL C00261 BC00261 V=666.7
COMM MOVL C00262 BC00262 V=166.7 PL=0
COMM REFP 3 C00263 BC00263
COMM CALL JOB:SEARCH-R1
COMM SET P0406 P0006
COMM SFTON P0406
COMM MOVL C00264 BC00264 V=166.7 PL=0
COMM REFP 3 C00265 BC00265
COMM CALL JOB:SEARCH-R1
COMM SET P0406 P0006
COMM SFTON P0406
COMM MOVL C00266 BC00266 V=250.0 PL=0
COMM SFTOF
COMM '------------------------
COMM 'W27.14
COMM '------------------------
COMM MOVL C00267 BC00267 V=666.7
COMM MOVL C00268 BC00268 V=100.0 PL=0
COMM REFP 3 C00269 BC00269
COMM CALL JOB:SEARCH-R1
COMM SET P0407 P0006
COMM SFTON P0407
COMM MOVL C00270 BC00270 V=166.7 PL=0
COMM REFP 3 C00271 BC00271
COMM CALL JOB:SEARCH-R1
COMM SET P0407 P0006
COMM SFTON P0407
COMM MOVL C00272 BC00272 V=250.0 PL=0
COMM SFTOF
COMM '------------------------
COMM 'W27.16
COMM '------------------------
COMM MOVL C00273 BC00273 V=666.7
COMM MOVL C00274 BC00274 V=100.0 PL=0
COMM REFP 3 C00275 BC00275
COMM CALL JOB:SEARCH-R1
COMM SET P0408 P0006
COMM SFTON P0408
COMM MOVL C00276 BC00276 V=166.7 PL=0
COMM REFP 3 C00277 BC00277
COMM CALL JOB:SEARCH-R1
COMM SET P0408 P0006
COMM SFTON P0408
COMM MOVL C00278 BC00278 V=250.0 PL=0
COMM MOVL C00279 BC00279 V=666.7
COMM SFTOF
COMM '------------------------
COMM 'W27.18
COMM '------------------------
COMM MOVJ C00280 BC00280 VJ=40.00
COMM MOVJ C00281 BC00281 VJ=50.00
COMM MOVL C00282 BC00282 V=666.7
COMM MOVL C00283 BC00283 V=333.3
COMM MOVL C00284 BC00284 V=100.0 PL=0
COMM REFP 3 C00285 BC00285
COMM CALL JOB:SEARCH-R1
COMM SET P0409 P0006
COMM SFTON P0409
COMM MOVL C00286 BC00286 V=16.7 PL=0
COMM REFP 3 C00287 BC00287
COMM CALL JOB:SEARCH-R1
COMM SET P0409 P0006
COMM SFTON P0409
COMM MOVL C00288 BC00288 V=166.7 PL=0
COMM SFTOF
COMM '------------------------
COMM 'W27.19
COMM '------------------------
COMM MOVL C00289 BC00289 V=666.7
COMM MOVL C00290 BC00290 V=100.0 PL=0
COMM REFP 3 C00291 BC00291
COMM CALL JOB:SEARCH-R1
COMM SET P0410 P0006
COMM SFTON P0410
COMM MOVL C00292 BC00292 V=166.7 PL=0
COMM REFP 3 C00293 BC00293
COMM CALL JOB:SEARCH-R1
COMM SET P0410 P0006
COMM SFTON P0410
COMM MOVL C00294 BC00294 V=250.0 PL=0
COMM SFTOF
COMM '------------------------
COMM 'W27.21
COMM '------------------------
COMM MOVL C00295 BC00295 V=666.7
COMM MOVL C00296 BC00296 V=133.3 PL=0
COMM REFP 3 C00297 BC00297
COMM CALL JOB:SEARCH-R1
COMM SET P0411 P0006
COMM SFTON P0411
COMM MOVL C00298 BC00298 V=166.7 PL=0
COMM REFP 3 C00299 BC00299
COMM CALL JOB:SEARCH-R1
COMM SET P0411 P0006
COMM SFTON P0411
COMM MOVL C00300 BC00300 V=166.7 PL=0
COMM SFTOF
COMM '------------------------
COMM 'W27.22
COMM '------------------------
COMM MOVL C00301 BC00301 V=666.7
COMM MOVL C00302 BC00302 V=100.0 PL=0
COMM REFP 3 C00303 BC00303
COMM CALL JOB:SEARCH-R1
COMM SET P0412 P0006
COMM SFTON P0412
COMM MOVL C00304 BC00304 V=166.7 PL=0
COMM REFP 3 C00305 BC00305
COMM CALL JOB:SEARCH-R1
COMM SET P0412 P0006
COMM SFTON P0412
COMM MOVL C00306 BC00306 V=166.7 PL=0
COMM SFTOF
COMM '------------------------
COMM 'W27.24
COMM '------------------------
COMM MOVL C00307 BC00307 V=666.7
COMM MOVL C00308 BC00308 V=100.0 PL=0
COMM REFP 3 C00309 BC00309
COMM CALL JOB:SEARCH-R1
COMM SET P0413 P0006
COMM SFTON P0413
COMM MOVL C00310 BC00310 V=166.7 PL=0
COMM REFP 3 C00311 BC00311
COMM CALL JOB:SEARCH-R1
COMM SET P0413 P0006
COMM SFTON P0413
COMM MOVL C00312 BC00312 V=250.0 PL=0
COMM SFTOF
COMM GETE D040 P0413 (1)
COMM GETE D041 P0413 (2)
COMM GETE D042 P0413 (3)
COMM SETE P0414 (1) D040
COMM SETE P0414 (2) D041
COMM SETE P0414 (3) D042
COMM GETE D040 P0413 (1)
COMM GETE D041 P0413 (2)
COMM GETE D042 P0413 (3)
COMM SETE P0415 (1) D040
COMM SETE P0415 (2) D041
COMM SETE P0415 (3) D042
COMM '------------------------
COMM 'W27.26
COMM '------------------------
COMM MOVL C00313 BC00313 V=333.3
COMM MOVL C00314 BC00314 V=66.7 PL=0
COMM REFP 3 C00315 BC00315
COMM CALL JOB:SEARCH-R1
COMM SET P0414 P0006
COMM SFTON P0414
COMM MOVL C00316 BC00316 V=66.7 PL=0
COMM REFP 3 C00317 BC00317
COMM CALL JOB:SEARCH-R1
COMM SET P0414 P0006
COMM SFTON P0414
COMM MOVL C00318 BC00318 V=66.7 PL=0
COMM SFTOF
COMM MOVL C00319 BC00319 V=333.3
COMM MOVL C00320 BC00320 V=666.7
COMM MOVL C00321 BC00321 V=1000.0
COMM MOVL C00322 BC00322 V=1000.0
COMM MOVL C00323 BC00323 V=666.7
COMM MOVL C00324 BC00324 V=500.0
COMM '------------------------
COMM 'W27.29
COMM '------------------------
COMM MOVL C00325 BC00325 V=333.3
COMM MOVL C00326 BC00326 V=100.0 PL=0
COMM REFP 3 C00327 BC00327
COMM CALL JOB:SEARCH-R1
COMM SET P0416 P0006
COMM SFTON P0416
COMM MOVL C00328 BC00328 V=166.7 PL=0
COMM REFP 3 C00329 BC00329
COMM CALL JOB:SEARCH-R1
COMM SET P0416 P0006
COMM SFTON P0416
COMM MOVL C00330 BC00330 V=250.0 PL=0
COMM SFTOF
COMM '------------------------
COMM 'W27.31
COMM '------------------------
COMM MOVL C00331 BC00331 V=666.7
COMM MOVL C00332 BC00332 V=100.0 PL=0
COMM REFP 3 C00333 BC00333
COMM CALL JOB:SEARCH-R1
COMM SET P0417 P0006
COMM SFTON P0417
COMM MOVL C00334 BC00334 V=166.7 PL=0
COMM REFP 3 C00335 BC00335
COMM CALL JOB:SEARCH-R1
COMM SET P0417 P0006
COMM SFTON P0417
COMM MOVL C00336 BC00336 V=250.0 PL=0
COMM SFTOF
COMM '------------------------
COMM 'W27.32
COMM '------------------------
COMM SFTOF
COMM MOVL C00337 BC00337 V=666.7
CALL JOB:FRONT_SEARCH_90ST-1_5540
MOVJ C00338 BC00338 VJ=50.00
MOVJ C00339 BC00339 VJ=40.00
MOVJ C00340 BC00340 VJ=40.00
MOVL C00341 BC00341 V=500.0
MOVJ C00342 BC00342 VJ=30.00
'------------------------
'W31.2
'------------------------
SFTON P0300
MOVL C00343 BC00343 V=500.0
MOVL C00344 BC00344 V=133.3 PL=0
MACRO1 MJ#(0) ARGF10
ARCON
MOVL C00345 BC00345 V=10.8
ARCOF
MOVL C00346 BC00346 V=250.0
SFTOF
'------------------------
'W31.4
'------------------------
SFTON P0301
MOVL C00347 BC00347 V=500.0
MOVL C00348 BC00348 V=166.7
MACRO1 MJ#(0) ARGF10
ARCON
MOVL C00349 BC00349 V=10.8
ARCOF
MOVL C00350 BC00350 V=250.0
SFTOF
'------------------------
'W31.6
'------------------------
SFTON P0302
MOVL C00351 BC00351 V=500.0
MOVL C00352 BC00352 V=166.7 PL=0
MACRO1 MJ#(0) ARGF10
ARCON
MOVL C00353 BC00353 V=10.8
ARCOF
MOVL C00354 BC00354 V=166.7
SFTOF
'------------------------
'W31.8
'------------------------
SFTON P0303
MOVL C00355 BC00355 V=500.0
MOVL C00356 BC00356 V=166.7 PL=0
MACRO1 MJ#(0) ARGF10
ARCON
MOVL C00357 BC00357 V=10.8
ARCOF
MOVL C00358 BC00358 V=166.7
SFTOF
'------------------------
'W31.9
'------------------------
SFTON P0304
MOVL C00359 BC00359 V=500.0
MOVL C00360 BC00360 V=166.7 PL=0
MACRO1 MJ#(0) ARGF10
ARCON
MOVL C00361 BC00361 V=10.8
ARCOF
MOVL C00362 BC00362 V=166.7
SFTOF
MOVL C00363 BC00363 V=500.0
MOVL C00364 BC00364 V=666.7
MOVJ C00365 BC00365 VJ=30.00
MOVJ C00366 BC00366 VJ=50.00
COMM '::::::::::::::::::::::::::::::::
COMM '::::::::::::::::::::::::::::::::
COMM '::::::::::::::::::::::::::::::::
COMM '::::::::::::::::::::::::::::::::
COMM '::::::::::::::::::::::::::::::::
COMM MOVJ C00367 BC00367 VJ=30.00
COMM MOVJ C00368 BC00368 VJ=30.00
COMM MOVJ C00369 BC00369 VJ=25.00
COMM MOVJ C00370 BC00370 VJ=30.00
COMM MOVJ C00371 BC00371 VJ=40.00
COMM '------------------------
COMM 'W27.1
COMM '------------------------
COMM MOVL C00372 BC00372 V=666.7
COMM SFTON P0401
COMM MOVL C00373 BC00373 V=166.7 PL=0
COMM MACRO1 MJ#(0) ARGF24
COMM ARCON
COMM MOVL C00374 BC00374 V=8.3
COMM ARCOF
COMM SFTOF
COMM 'BELKA PRZEJAZD
COMM MOVL C00375 BC00375 V=250.0
COMM MOVL C00376 BC00376 V=333.3
COMM SFTON P0402
COMM MOVL C00377 BC00377 V=166.7
COMM ARCON
COMM MOVL C00378 BC00378 V=8.3
COMM ARCOF
COMM SFTOF
COMM MOVL C00379 BC00379 V=166.7
COMM MOVL C00380 BC00380 V=333.3
COMM SFTON P0403
COMM MOVL C00381 BC00381 V=166.7
COMM ARCON
COMM MOVL C00382 BC00382 V=8.3
COMM ARCOF
COMM SFTOF
COMM MOVL C00383 BC00383 V=250.0
COMM MOVJ C00384 BC00384 VJ=30.00
COMM MOVJ C00385 BC00385 VJ=30.00
COMM MOVJ C00386 BC00386 VJ=40.00
MOVJ C00387 BC00387 VJ=50.00
MOVJ C00388 BC00388 VJ=50.00
MOVJ C00389 BC00389 VJ=50.00
MOVL C00390 BC00390 V=166.7
'------------------------
'W213A
'------------------------
SFTON P0355
MOVL C00391 BC00391 V=500.0
MOVL C00392 BC00392 V=166.7 PL=0
MACRO1 MJ#(0) ARGF9
ARCON
SFTOF
SFTON P0354
MOVL C00393 BC00393 V=11.7
ARCOF
MOVL C00394 BC00394 V=166.7
SFTOF
MOVJ C00395 BC00395 VJ=50.00
MOVJ C00396 BC00396 VJ=80.00
MOVJ C00397 BC00397 VJ=10.00
MOVJ C00398 BC00398 VJ=40.00
MOVJ C00399 BC00399 VJ=40.00
MOVJ C00400 BC00400 VJ=30.00
MOVJ C00401 BC00401 VJ=30.00
'5.5.1
'------------------------
'W31.11
'------------------------
SFTON P0305
MOVL C00402 BC00402 V=333.3
MOVL C00403 BC00403 V=166.7
MACRO1 MJ#(0) ARGF10
ARCON
MOVL C00404 BC00404 V=10.8
ARCOF
MOVL C00405 BC00405 V=166.7
SFTOF
'------------------------
'W31.13
'------------------------
SFTON P0306
MOVL C00406 BC00406 V=333.3
MOVL C00407 BC00407 V=166.7
ARCON
MOVL C00408 BC00408 V=10.8
ARCOF
MOVL C00409 BC00409 V=166.7
SFTOF
'------------------------
'W31.14
'------------------------
SFTON P0307
MOVL C00410 BC00410 V=333.3
MOVL C00411 BC00411 V=166.7 PL=0
ARCON
MOVL C00412 BC00412 V=10.8
ARCOF
MOVL C00413 BC00413 V=250.0
SFTOF
MOVL C00414 BC00414 V=500.0
MOVL C00415 BC00415 V=500.0
SFTON P0309
MOVL C00416 BC00416 V=166.7
ARCON
MOVL C00417 BC00417 V=10.8
ARCOF
SFTOF
MOVL C00418 BC00418 V=166.7
MOVL C00419 BC00419 V=500.0
MOVJ C00420 BC00420 VJ=30.00
MOVJ C00421 BC00421 VJ=30.00
MOVJ C00422 BC00422 VJ=30.00
MOVJ C00423 BC00423 VJ=40.00
COMM '::::::::::::::::::::::::::::::::
COMM '::::::::::::::::::::::::::::::::
COMM '------------------------
COMM 'W27.9
COMM '------------------------
COMM '::::::::::::::::::::::::::::::::
COMM '::::::::::::::::::::::::::::::::
COMM MOVJ C00424 BC00424 VJ=40.00
COMM MOVJ C00425 BC00425 VJ=30.00
COMM MOVL C00426 BC00426 V=666.7
COMM SFTON P0404
COMM MOVL C00427 BC00427 V=500.0
COMM MOVL C00428 BC00428 V=200.0 PL=0
COMM MACRO1 MJ#(0) ARGF24
COMM ARCON
COMM MOVL C00429 BC00429 V=7.5
COMM ARCOF
COMM MOVL C00430 BC00430 V=166.7
COMM SFTOF
COMM MOVL C00431 BC00431 V=500.0
COMM MOVL C00432 BC00432 V=500.0
COMM MOVJ C00433 BC00433 VJ=50.00
COMM MOVJ C00434 BC00434 VJ=50.00
COMM '------------------------
COMM 'W27.11
COMM MACRO1 MJ#(0) ARGF24
COMM '------------------------
COMM MOVL C00435 BC00435 V=500.0
COMM SFTON P0404
COMM MOVL C00436 BC00436 V=250.0
COMM ARCON
COMM MOVL C00437 BC00437 V=8.3
COMM ARCOF
COMM SFTOF
COMM SFTON P0405
COMM MOVL C00438 BC00438 V=333.3
COMM MOVL C00439 BC00439 V=200.0 PL=0
COMM ARCON
COMM MOVL C00440 BC00440 V=8.3
COMM ARCOF
COMM MOVL C00441 BC00441 V=166.7
COMM SFTOF
COMM MOVL C00442 BC00442 V=416.7
'------------------------
COMM 'W27.13
COMM '------------------------
COMM SFTON P0406
COMM MOVL C00443 BC00443 V=333.3
COMM MOVL C00444 BC00444 V=133.3 PL=0
COMM MACRO1 MJ#(0) ARGF24
COMM ARCON
COMM MOVL C00445 BC00445 V=7.5
COMM ARCOF
COMM MOVL C00446 BC00446 V=250.0
SFTOF
COMM MOVJ C00447 BC00447 VJ=50.00
COMM MOVJ C00448 BC00448 VJ=50.00
COMM MOVJ C00449 BC00449 VJ=50.00
'::::::::::::::::::::::::
'::::::::::::::::::::::::
'::::::::::::::::::::::::
'::::::::::::::::::::::::
'::::::::::::::::::::::::
'::::::::::::::::::::::::
'::::::::::::::::::::::::
MOVJ C00450 BC00450 VJ=50.00
MOVJ C00451 BC00451 VJ=30.00
'------------------------
'W214A
'------------------------
SFTON P0351
MOVL C00452 BC00452 V=333.3
MOVL C00453 BC00453 V=500.0
MOVL C00454 BC00454 V=166.7 PL=0
MACRO1 MJ#(0) ARGF9
ARCON
SFTOF
SFTON P0350
MOVL C00455 BC00455 V=11.7
ARCOF
MOVL C00456 BC00456 V=250.0
SFTOF
MOVJ C00457 BC00457 VJ=50.00
MOVJ C00458 BC00458 VJ=50.00
MOVJ C00459 BC00459 VJ=10.00
MOVJ C00460 BC00460 VJ=50.00
MOVJ C00461 BC00461 VJ=50.00
MOVJ C00462 BC00462 VJ=50.00
MOVJ C00463 BC00463 VJ=30.00
MOVJ C00464 BC00464 VJ=20.00
'------------------------
'W31.16
MACRO1 MJ#(0) ARGF10
'------------------------
SFTON P0308
MOVL C00465 BC00465 V=333.3
MOVL C00466 BC00466 V=66.7 PL=0
ARCON
MOVL C00467 BC00467 V=10.8
ARCOF
SFTOF
MOVL C00468 BC00468 V=250.0
SFTOF
MOVL C00469 BC00469 V=500.0
MOVL C00470 BC00470 V=500.0
MOVL C00471 BC00471 V=500.0
MOVL C00472 BC00472 V=666.7
MOVL C00473 BC00473 V=833.3
MOVL C00474 BC00474 V=666.7
MOVL C00475 BC00475 V=333.3
MOVL C00476 BC00476 V=333.3
'------------------------
'W31.18
'------------------------
SFTON P0310
MOVL C00477 BC00477 V=166.7 PL=0
ARCON
MOVL C00478 BC00478 V=10.8
ARCOF
MOVL C00479 BC00479 V=166.7
SFTOF
'------------------------
'W31.19
'------------------------
SFTOF
MOVL C00480 BC00480 V=500.0
MOVL C00481 BC00481 V=666.7
MOVL C00482 BC00482 V=666.7
MOVJ C00483 BC00483 VJ=50.00
COMM '::::::::::::::::::::::::
COMM '::::::::::::::::::::::::
COMM '::::::::::::::::::::::::
COMM '::::::::::::::::::::::::
COMM '::::::::::::::::::::::::
COMM '::::::::::::::::::::::::
COMM '::::::::::::::::::::::::
COMM MOVJ C00484 BC00484 VJ=50.00
COMM MOVJ C00485 BC00485 VJ=40.00
COMM '::::::::::::::::::::::::::::::::
COMM '::::::::::::::::::::::::::::::::
COMM '------------------------
COMM 'W27.14
COMM '------------------------
COMM '::::::::::::::::::::::::::::::::
COMM '::::::::::::::::::::::::::::::::
COMM SFTON P0407
COMM MOVJ C00486 BC00486 VJ=40.00
COMM MOVL C00487 BC00487 V=500.0
COMM MOVL C00488 BC00488 V=166.7 PL=0
COMM MACRO1 MJ#(0) ARGF24
COMM ARCON
COMM MOVL C00489 BC00489 V=7.5
COMM ARCOF
COMM MOVL C00490 BC00490 V=250.0
COMM SFTOF
COMM '------------------------
COMM 'W27.16
COMM '------------------------
COMM SFTON P0408
COMM MOVL C00491 BC00491 V=333.3
COMM MOVL C00492 BC00492 V=166.7 PL=0
COMM MACRO1 MJ#(0) ARGF24
COMM ARCON
COMM MOVL C00493 BC00493 V=7.5
COMM ARCOF
COMM MOVL C00494 BC00494 V=250.0
COMM SFTOF
COMM MOVL C00495 BC00495 V=500.0
COMM MOVL C00496 BC00496 V=500.0
COMM MOVJ C00497 BC00497 VJ=40.00
COMM MOVJ C00498 BC00498 VJ=40.00
COMM MOVL C00499 BC00499 V=666.7
COMM '------------------------
COMM 'W27.18
COMM '------------------------
COMM SFTON P0409
COMM MOVL C00500 BC00500 V=500.0
COMM MOVL C00501 BC00501 V=166.7 PL=0
COMM MACRO1 MJ#(0) ARGF24
COMM ARCON
COMM MOVL C00502 BC00502 V=7.5
COMM ARCOF
COMM MOVL C00503 BC00503 V=250.0
COMM SFTOF
COMM MOVJ C00504 BC00504 VJ=20.00
COMM MOVJ C00505 BC00505 VJ=30.00
COMM MOVJ C00506 BC00506 VJ=50.00
COMM '::::::::::::::::::::::::
COMM '::::::::::::::::::::::::
COMM '::::::::::::::::::::::::
COMM '::::::::::::::::::::::::
COMM '::::::::::::::::::::::::
COMM '::::::::::::::::::::::::
COMM '::::::::::::::::::::::::
MOVJ C00507 BC00507 VJ=50.00
MOVJ C00508 BC00508 VJ=50.00
'------------------------
'W215A
'------------------------
SFTON P0359
MOVL C00509 BC00509 V=666.7
MOVL C00510 BC00510 V=166.7 PL=0
MACRO1 MJ#(0) ARGF9
ARCON
SFTOF
SFTON P0358
MOVL C00511 BC00511 V=11.7
ARCOF
MOVL C00512 BC00512 V=333.3
SFTOF
MOVJ C00513 BC00513 VJ=30.00
MOVJ C00514 BC00514 VJ=50.00
MOVJ C00515 BC00515 VJ=50.00
MOVJ C00516 BC00516 VJ=50.00
MOVJ C00517 BC00517 VJ=50.00
MOVJ C00518 BC00518 VJ=50.00
MOVJ C00519 BC00519 VJ=30.00
MOVJ C00520 BC00520 VJ=30.00
'------------------------
'W31.21
'------------------------
SFTON P0311
MOVL C00521 BC00521 V=666.7
MOVL C00522 BC00522 V=166.7 PL=0
MACRO1 MJ#(0) ARGF10
ARCON
MOVL C00523 BC00523 V=10.8
ARCOF
MOVL C00524 BC00524 V=250.0
SFTOF
'------------------------
'W31.22
'------------------------
SFTON P0312
MOVL C00525 BC00525 V=333.3
MOVL C00526 BC00526 V=166.7 PL=0
ARCON
MOVL C00527 BC00527 V=10.8
ARCOF
MOVL C00528 BC00528 V=250.0
SFTOF
'------------------------
'W31.24
'------------------------
SFTON P0313
MOVL C00529 BC00529 V=500.0
MOVL C00530 BC00530 V=166.7 PL=0
MACRO1 MJ#(0) ARGF10
ARCON
MOVL C00531 BC00531 V=10.8
ARCOF
MOVL C00532 BC00532 V=250.0
MOVL C00533 BC00533 V=333.3
MOVL C00534 BC00534 V=500.0
SFTOF
MOVL C00535 BC00535 V=666.7
MOVJ C00536 BC00536 VJ=50.00
MOVJ C00537 BC00537 VJ=50.00
MOVJ C00538 BC00538 VJ=50.00
'::::::::::::::::::::::::
'::::::::::::::::::::::::
'::::::::::::::::::::::::
'::::::::::::::::::::::::
'::::::::::::::::::::::::
'::::::::::::::::::::::::
'::::::::::::::::::::::::
MOVJ C00539 BC00539 VJ=50.00
COMM MOVJ C00540 BC00540 VJ=30.00
COMM MOVJ C00541 BC00541 VJ=30.00
COMM MOVJ C00542 BC00542 VJ=30.00
COMM '::::::::::::::::::::::::::::::::
COMM '::::::::::::::::::::::::::::::::
COMM '------------------------
COMM 'W27.19
COMM '------------------------
COMM '::::::::::::::::::::::::::::::::
COMM '::::::::::::::::::::::::::::::::
COMM SFTOF
COMM MOVL C00543 BC00543 V=666.7
COMM MOVL C00544 BC00544 V=666.7
COMM MOVL C00545 BC00545 V=666.7
COMM SFTON P0410
COMM MOVL C00546 BC00546 V=166.7 PL=0
COMM MACRO1 MJ#(0) ARGF24
COMM ARCON
COMM MOVL C00547 BC00547 V=7.5
COMM ARCOF
COMM MOVL C00548 BC00548 V=333.3
COMM SFTOF
COMM MOVJ C00549 BC00549 VJ=30.00
COMM MOVJ C00550 BC00550 VJ=50.00
COMM MOVJ C00551 BC00551 VJ=50.00
COMM MOVJ C00552 BC00552 VJ=50.00
COMM MOVJ C00553 BC00553 VJ=50.00
COMM MOVJ C00554 BC00554 VJ=30.00
COMM '------------------------
COMM 'W27.21
COMM '------------------------
COMM SFTON P0411
COMM MOVL C00555 BC00555 V=333.3
COMM MOVL C00556 BC00556 V=166.7 PL=0
COMM MACRO1 MJ#(0) ARGF24
COMM ARCON
COMM MOVL C00557 BC00557 V=7.5
COMM ARCOF
COMM MOVL C00558 BC00558 V=333.3
COMM SFTOF
COMM '------------------------
COMM 'W27.22
COMM '------------------------
COMM SFTON P0412
COMM MOVL C00559 BC00559 V=333.3
COMM MOVL C00560 BC00560 V=166.7 PL=0
COMM MACRO1 MJ#(0) ARGF24
COMM ARCON
COMM MOVL C00561 BC00561 V=7.5
COMM ARCOF
COMM SFTOF
COMM MOVL C00562 BC00562 V=250.0
COMM SFTOF
COMM '::::::::::::::::::::::::
COMM '::::::::::::::::::::::::
COMM '::::::::::::::::::::::::
COMM '::::::::::::::::::::::::
COMM '::::::::::::::::::::::::
COMM '::::::::::::::::::::::::
COMM '::::::::::::::::::::::::
COMM MOVJ C00563 BC00563 VJ=30.00
COMM MOVJ C00564 BC00564 VJ=40.00
COMM MOVJ C00565 BC00565 VJ=80.00
COMM MOVJ C00566 BC00566 VJ=80.00
'------------------------
'W215A
'------------------------
MOVJ C00567 BC00567 VJ=80.00
MOVJ C00568 BC00568 VJ=80.00
SFTON P0360
MOVL C00569 BC00569 V=500.0
MOVL C00570 BC00570 V=666.7
MOVL C00571 BC00571 V=166.7 PL=0
MACRO1 MJ#(0) ARGF9
ARCON
SFTOF
SFTON P0361
MOVL C00572 BC00572 V=11.7
ARCOF
MOVL C00573 BC00573 V=333.3
SFTOF
MOVJ C00574 BC00574 VJ=50.00
MOVJ C00575 BC00575 VJ=50.00
MOVJ C00576 BC00576 VJ=50.00
MOVJ C00577 BC00577 VJ=60.00
MOVJ C00578 BC00578 VJ=50.00
MOVJ C00579 BC00579 VJ=50.00
MOVJ C00580 BC00580 VJ=30.00
'------------------------
'W31.26
'------------------------
SFTON P0314
MOVL C00581 BC00581 V=666.7
MOVL C00582 BC00582 V=166.7 PL=0
MACRO1 MJ#(0) ARGF10
ARCON
MOVL C00583 BC00583 V=10.8
ARCOF
MOVL C00584 BC00584 V=166.7
SFTOF
'------------------------
'W31.27
'------------------------
SFTON P0315
MOVL C00585 BC00585 V=166.7 PL=0
MACRO1 MJ#(0) ARGF10
ARCON
MOVL C00586 BC00586 V=10.8
ARCOF
MOVL C00587 BC00587 V=250.0
SFTOF
SFTOF
MOVL C00588 BC00588 V=333.3
MOVL C00589 BC00589 V=333.3
MOVL C00590 BC00590 V=333.3
MOVJ C00591 BC00591 VJ=50.00
MOVJ C00592 BC00592 VJ=50.00
MOVJ C00593 BC00593 VJ=40.00
MOVJ C00594 BC00594 VJ=50.00
COMM '::::::::::::::::::::::::
COMM '::::::::::::::::::::::::
COMM '::::::::::::::::::::::::
COMM '::::::::::::::::::::::::
COMM '::::::::::::::::::::::::
COMM '::::::::::::::::::::::::
COMM '::::::::::::::::::::::::
COMM MOVJ C00595 BC00595 VJ=50.00
COMM MOVJ C00596 BC00596 VJ=50.00
COMM '::::::::::::::::::::::::::::::::
COMM '::::::::::::::::::::::::::::::::
COMM '------------------------
COMM 'W27.24
COMM '------------------------
COMM '::::::::::::::::::::::::::::::::
COMM '::::::::::::::::::::::::::::::::
COMM SFTON P0413
COMM MOVL C00597 BC00597 V=666.7
COMM MOVL C00598 BC00598 V=166.7 PL=0
COMM MACRO1 MJ#(0) ARGF24
COMM ARCON
COMM MOVL C00599 BC00599 V=7.5
COMM ARCOF
COMM MOVL C00600 BC00600 V=250.0
COMM SFTOF
COMM '------------------------
COMM 'W27.26
COMM '------------------------
COMM SFTON P0414
COMM MOVL C00601 BC00601 V=333.3
COMM MOVL C00602 BC00602 V=166.7 PL=0
COMM MACRO1 MJ#(0) ARGF24
COMM ARCON
COMM MOVL C00603 BC00603 V=7.5
COMM ARCOF
COMM MOVL C00604 BC00604 V=250.0
COMM SFTOF
COMM '------------------------
COMM 'W27.27
COMM '------------------------
COMM SFTON P0414
COMM MOVL C00605 BC00605 V=333.3
COMM MOVL C00606 BC00606 V=66.7 PL=0
COMM MACRO1 MJ#(0) ARGF24
COMM ARCON
COMM MOVL C00607 BC00607 V=6.7
COMM ARCOF
COMM MOVL C00608 BC00608 V=83.3
COMM SFTOF
COMM MOVL C00609 BC00609 V=333.3
COMM '::::::::::::::::::::::::
COMM '::::::::::::::::::::::::
COMM '::::::::::::::::::::::::
COMM '::::::::::::::::::::::::
COMM '::::::::::::::::::::::::
COMM '::::::::::::::::::::::::
COMM '::::::::::::::::::::::::
COMM MOVL C00610 BC00610 V=666.7
COMM MOVJ C00611 BC00611 VJ=40.00
COMM MOVJ C00612 BC00612 VJ=40.00
COMM MOVJ C00613 BC00613 VJ=40.00
COMM MOVJ C00614 BC00614 VJ=40.00
COMM '------------------------
COMM 'W218A
COMM '------------------------
MOVJ C00615 BC00615 VJ=50.00
MOVJ C00616 BC00616 VJ=50.00
SFTON P0357
MOVL C00617 BC00617 V=666.7
MOVL C00618 BC00618 V=166.7 PL=0
MACRO1 MJ#(0) ARGF9
ARCON
SFTOF
SFTON P0356
MOVL C00619 BC00619 V=11.7
ARCOF
MOVL C00620 BC00620 V=333.3
MOVL C00621 BC00621 V=500.0
SFTOF
MOVJ C00622 BC00622 VJ=50.00
MOVJ C00623 BC00623 VJ=50.00
MOVJ C00624 BC00624 VJ=50.00
MOVJ C00625 BC00625 VJ=50.00
MOVJ C00626 BC00626 VJ=50.00
MOVJ C00627 BC00627 VJ=30.00
MOVL C00628 BC00628 V=666.7
'------------------------
'W31.29
'------------------------
SFTON P0316
MOVL C00629 BC00629 V=333.3
MOVL C00630 BC00630 V=333.3
MOVL C00631 BC00631 V=133.3 PL=0
MACRO1 MJ#(0) ARGF10
ARCON
MOVL C00632 BC00632 V=10.8
ARCOF
MOVL C00633 BC00633 V=250.0
SFTOF
MOVL C00634 BC00634 V=333.3
'------------------------
MOVL C00635 BC00635 V=333.3
MOVL C00636 BC00636 V=333.3
MOVL C00637 BC00637 V=333.3
MOVL C00638 BC00638 V=333.3
'W31.31
'------------------------
SFTON P0317
MOVL C00639 BC00639 V=666.7
MOVL C00640 BC00640 V=166.7 PL=0
ARCON
MOVL C00641 BC00641 V=10.8
ARCOF
MOVL C00642 BC00642 V=250.0
SFTOF
'------------------------
'W31.32
'------------------------
SFTON P0317
MOVL C00643 BC00643 V=333.3 PL=0
MOVL C00644 BC00644 V=166.7 PL=0
ARCON
MOVL C00645 BC00645 V=10.8
ARCOF
MOVL C00646 BC00646 V=250.0
SFTOF
MOVL C00647 BC00647 V=333.3
MOVL C00648 BC00648 V=333.3
SFTON P0320
MOVL C00649 BC00649 V=166.7
ARCON
MOVL C00650 BC00650 V=10.8
ARCOF
SFTOF
MOVL C00651 BC00651 V=250.0
MOVL C00652 BC00652 V=333.3
MOVL C00653 BC00653 V=333.3
MOVL C00654 BC00654 V=500.0
MOVL C00655 BC00655 V=500.0
MOVL C00656 BC00656 V=500.0
MOVJ C00657 BC00657 VJ=40.00
MOVJ C00658 BC00658 VJ=40.00
COMM MOVJ C00659 BC00659 VJ=40.00
COMM MOVJ C00660 BC00660 VJ=40.00
COMM '::::::::::::::::::::::::
COMM '::::::::::::::::::::::::
COMM '::::::::::::::::::::::::
COMM '::::::::::::::::::::::::
COMM '::::::::::::::::::::::::
COMM '::::::::::::::::::::::::
COMM '::::::::::::::::::::::::
COMM MOVJ C00661 BC00661 VJ=40.00
COMM MOVJ C00662 BC00662 VJ=40.00
COMM MOVJ C00663 BC00663 VJ=40.00
COMM '::::::::::::::::::::::::::::::::
COMM '::::::::::::::::::::::::::::::::
COMM '------------------------
COMM 'W27.29
COMM '------------------------
COMM '::::::::::::::::::::::::::::::::
COMM '::::::::::::::::::::::::::::::::
COMM SFTON P0416
COMM MOVL C00664 BC00664 V=500.0
COMM MOVL C00665 BC00665 V=166.7 PL=0
COMM MACRO1 MJ#(0) ARGF24
COMM ARCON
COMM MOVL C00666 BC00666 V=7.5
COMM ARCOF
COMM MOVL C00667 BC00667 V=250.0
COMM MOVL C00668 BC00668 V=250.0
COMM SFTON P0416
COMM MOVL C00669 BC00669 V=166.7
COMM ARCON
COMM MOVL C00670 BC00670 V=7.5
COMM ARCOF
COMM SFTOF
COMM MOVL C00671 BC00671 V=166.7
COMM '------------------------
COMM 'W27.31
COMM '------------------------
COMM SFTOF
COMM '::::::::::::::::::::::::
COMM '::::::::::::::::::::::::
COMM '::::::::::::::::::::::::
COMM '::::::::::::::::::::::::
COMM '::::::::::::::::::::::::
COMM '::::::::::::::::::::::::
COMM '::::::::::::::::::::::::
COMM MOVL C00672 BC00672 V=500.0
COMM MOVJ C00673 BC00673 VJ=50.00
COMM MOVJ C00674 BC00674 VJ=50.00
COMM MOVJ C00675 BC00675 VJ=50.00
COMM MOVJ C00676 BC00676 VJ=50.00
COMM MOVJ C00677 BC00677 VJ=50.00
COMM '------------------------
COMM 'W219A
COMM '------------------------
COMM MOVJ C00678 BC00678 VJ=50.00
MOVJ C00679 BC00679 VJ=50.00
SFTON P0353
MOVL C00680 BC00680 V=500.0
MOVL C00681 BC00681 V=333.3
MOVL C00682 BC00682 V=166.7 PL=0
MACRO1 MJ#(0) ARGF9
ARCON
SFTOF
SFTON P0352
MOVL C00683 BC00683 V=11.7
ARCOF
MOVL C00684 BC00684 V=250.0
SFTOF
MOVJ C00685 BC00685 VJ=40.00
MOVJ C00686 BC00686 VJ=50.00
CALL JOB:FRONT_WELD_90ST-1_5540
CALL JOB:MOVE_OUT_OF_TUNNEL
END
